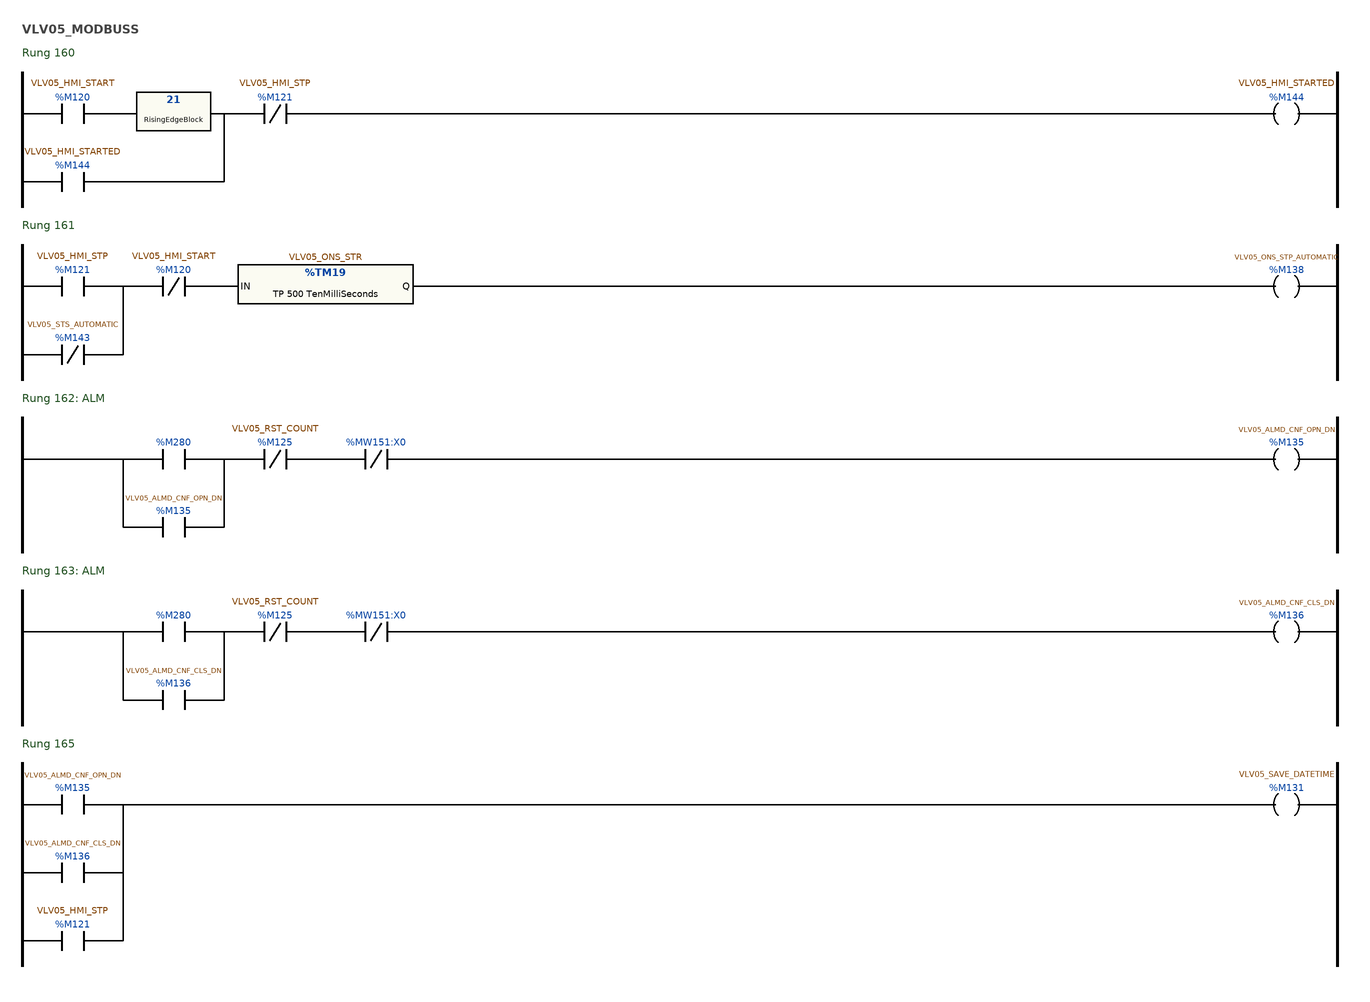
[picture p24: VLV05_MODBUSS, ladder]

// Rung 160
  LD %M120                (* VLV05_HMI_START *)
  RISING21
  OR %M144                (* VLV05_HMI_STARTED *)
  ANDN %M121              (* VLV05_HMI_STP *)
  ST %M144                (* VLV05_HMI_STARTED *)
  // as ST:
  //   VLV05_HMI_STARTED := (RISING(VLV05_HMI_START) OR VLV05_HMI_STARTED) AND NOT VLV05_HMI_STP;

// Rung 161
  BLK %TM19               (* VLV05_ONS_STR *)
  LD %M121                (* VLV05_HMI_STP *)
  ORN %M143               (* VLV05_STS_AUTOMATIC *)
  ANDN %M120              (* VLV05_HMI_START *)
  IN
  OUT_BLK
  LD Q
  ST %M138                (* VLV05_ONS_STP_AUTOMATIC *)
  END_BLK
  // as ST:
  //   VLV05_ONS_STR(IN := (VLV05_HMI_STP OR NOT VLV05_STS_AUTOMATIC) AND NOT VLV05_HMI_START);
  //   VLV05_ONS_STP_AUTOMATIC := VLV05_ONS_STR.Q;

// Rung 162: ALM
  LD 1
  AND( %M280
  OR %M135                (* VLV05_ALMD_CNF_OPN_DN *)
  )
  ANDN %M125              (* VLV05_RST_COUNT *)
  ANDN %MW151:X0
  ST %M135                (* VLV05_ALMD_CNF_OPN_DN *)
  // as ST:
  //   VLV05_ALMD_CNF_OPN_DN := (%M280 OR VLV05_ALMD_CNF_OPN_DN) AND NOT VLV05_RST_COUNT AND NOT %MW151:X0;

// Rung 163: ALM
  LD 1
  AND( %M280
  OR %M136                (* VLV05_ALMD_CNF_CLS_DN *)
  )
  ANDN %M125              (* VLV05_RST_COUNT *)
  ANDN %MW151:X0
  ST %M136                (* VLV05_ALMD_CNF_CLS_DN *)
  // as ST:
  //   VLV05_ALMD_CNF_CLS_DN := (%M280 OR VLV05_ALMD_CNF_CLS_DN) AND NOT VLV05_RST_COUNT AND NOT %MW151:X0;

// Rung 164
  LD 1
  MULTIFB
  LD 1
  AND %M21                (* HORARIOOFICINA_ACTIVE *)
  AND %M144               (* VLV05_HMI_STARTED *)
  ANDN %M135              (* VLV05_ALMD_CNF_OPN_DN *)
  ANDN %M136              (* VLV05_ALMD_CNF_CLS_DN *)
  AND %MW444:X0
  ANDN %M148              (* VLV05_TON_HR_DN *)
  ST %MW2509:X0
  LD %MW2509:X0
  ST %M143                (* VLV05_STS_AUTOMATIC *)
  BLK %TM47               (* VLV05_ONS_01 *)
  LD %MW2509:X0
  IN
  OUT_BLK
  LD Q
  ST %M126                (* VLV05_ONS_STS_AUTOMATIC *)
  END_BLK
  MULTIFB
  // as ST:
  //   %MW2509:X0 := HORARIOOFICINA_ACTIVE AND VLV05_HMI_STARTED AND NOT VLV05_ALMD_CNF_OPN_DN AND NOT VLV05_ALMD_CNF_CLS_DN AND %MW444:X0 AND NOT VLV05_TON_HR_DN;
  //   VLV05_STS_AUTOMATIC := %MW2509:X0;
  //   VLV05_ONS_01(IN := %MW2509:X0);
  //   VLV05_ONS_STS_AUTOMATIC := VLV05_ONS_01.Q;
  (* the ladder stored for this rung does not match its IL; not drawn *)

// Rung 165
  LD %M135                (* VLV05_ALMD_CNF_OPN_DN *)
  OR %M136                (* VLV05_ALMD_CNF_CLS_DN *)
  OR %M121                (* VLV05_HMI_STP *)
  ST %M131                (* VLV05_SAVE_DATETIME *)
  // as ST:
  //   VLV05_SAVE_DATETIME := VLV05_ALMD_CNF_OPN_DN OR VLV05_ALMD_CNF_CLS_DN OR VLV05_HMI_STP;

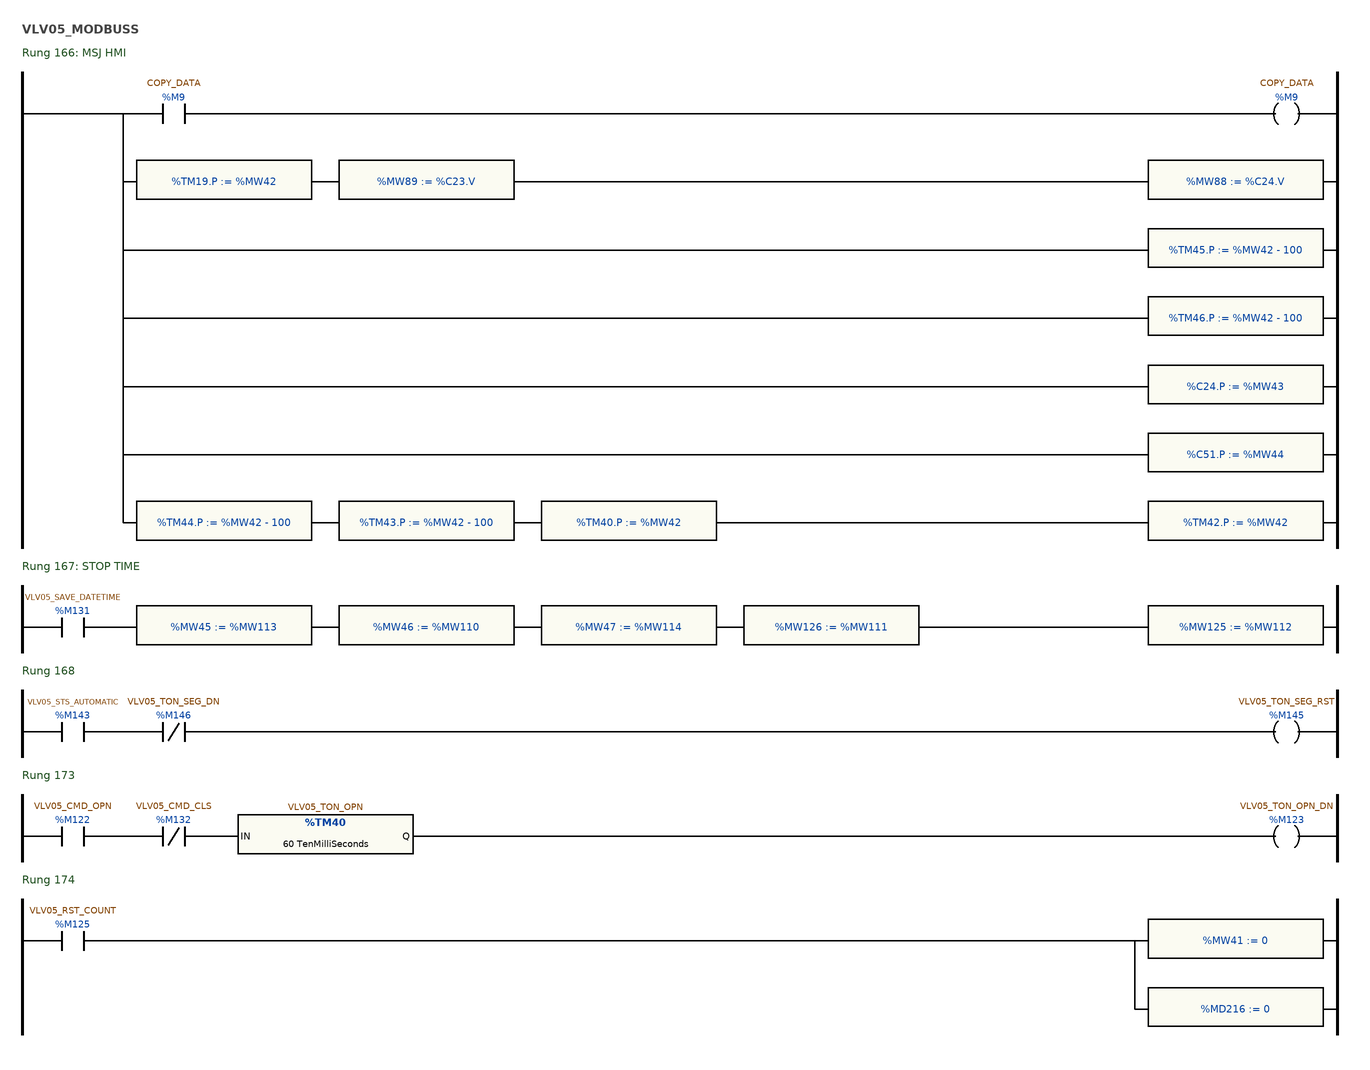

// Rung 166: MSJ HMI
  LD 1
  MPS
  AND %M9                 (* COPY_DATA *)
  ST %M9                  (* COPY_DATA *)
  MRD
  OPER [ %TM19.P := %MW42 ](* VLV05_ONS_STR, VLV05_T_CNF_PRESET *)
  OPER [ %MW89 := %C23.V ](* VLV05_CNT_MIN *)
  [ %MW88 := %C24.V ]     (* VLV05_CNT_HR *)
  MRD
  [ %TM45.P := %MW42 - 100 ](* VLV05_T_CNF_OPN, VLV05_T_CNF_PRESET *)
  MRD
  [ %TM46.P := %MW42 - 100 ](* VLV05_T_CNF_CLS, VLV05_T_CNF_PRESET *)
  MRD
  [ %C24.P := %MW43 ]     (* VLV05_CNT_HR, VLV05_CNF_HR_PRESET *)
  MRD
  [ %C51.P := %MW44 ]
  MPP
  OPER [ %TM44.P := %MW42 - 100 ](* VLV05_TON_ALMD_CNF_CLS, VLV05_T_CNF_PRESET *)
  OPER [ %TM43.P := %MW42 - 100 ](* VLV05_TON_ALMD_CNF_OPN, VLV05_T_CNF_PRESET *)
  OPER [ %TM40.P := %MW42 ](* VLV05_TON_OPN, VLV05_T_CNF_PRESET *)
  [ %TM42.P := %MW42 ]    (* VLV05_TON_CLS, VLV05_T_CNF_PRESET *)
  // as ST:
  //   COPY_DATA := COPY_DATA;
  //   VLV05_ONS_STR.P := VLV05_T_CNF_PRESET;
  //   %MW89 := VLV05_CNT_MIN.V;
  //   %MW88 := VLV05_CNT_HR.V;
  //   VLV05_T_CNF_OPN.P := VLV05_T_CNF_PRESET - 100;
  //   VLV05_T_CNF_CLS.P := VLV05_T_CNF_PRESET - 100;
  //   VLV05_CNT_HR.P := VLV05_CNF_HR_PRESET;
  //   %C51.P := %MW44;
  //   VLV05_TON_ALMD_CNF_CLS.P := VLV05_T_CNF_PRESET - 100;
  //   VLV05_TON_ALMD_CNF_OPN.P := VLV05_T_CNF_PRESET - 100;
  //   VLV05_TON_OPN.P := VLV05_T_CNF_PRESET;
  //   VLV05_TON_CLS.P := VLV05_T_CNF_PRESET;

// Rung 167: STOP TIME
  LD %M131                (* VLV05_SAVE_DATETIME *)
  OPER [ %MW45 := %MW113 ](* VLV05_RTC_HHMM, MONTH *)
  OPER [ %MW46 := %MW110 ](* VLV05_RTC_MMDD, DAY *)
  OPER [ %MW47 := %MW114 ](* VLV05_RTC_YY, YEAR *)
  OPER [ %MW126 := %MW111 ](* HOUR *)
  [ %MW125 := %MW112 ]    (* MINUTES *)
  // as ST:
  //   IF VLV05_SAVE_DATETIME THEN VLV05_RTC_HHMM := MONTH; END_IF;
  //   IF VLV05_SAVE_DATETIME THEN VLV05_RTC_MMDD := DAY; END_IF;
  //   IF VLV05_SAVE_DATETIME THEN VLV05_RTC_YY := YEAR; END_IF;
  //   IF VLV05_SAVE_DATETIME THEN %MW126 := HOUR; END_IF;
  //   IF VLV05_SAVE_DATETIME THEN %MW125 := MINUTES; END_IF;

// Rung 168
  LD %M143                (* VLV05_STS_AUTOMATIC *)
  ANDN %M146              (* VLV05_TON_SEG_DN *)
  ST %M145                (* VLV05_TON_SEG_RST *)
  // as ST:
  //   VLV05_TON_SEG_RST := VLV05_STS_AUTOMATIC AND NOT VLV05_TON_SEG_DN;

// Rung 169
  BLK %C24                (* VLV05_CNT_HR *)
  LD %M125                (* VLV05_RST_COUNT *)
  OR( %M21                (* HORARIOOFICINA_ACTIVE *)
  RISING22
  )
  R
  LD %M147                (* VLV05_TON_MIN_DN *)
  CU
  OUT_BLK
  LD D
  ST %M148                (* VLV05_TON_HR_DN *)
  END_BLK
  // as ST:
  //   VLV05_CNT_HR(RISING22 := HORARIOOFICINA_ACTIVE, R := VLV05_RST_COUNT OR HORARIOOFICINA_ACTIVE, CU := VLV05_TON_MIN_DN);
  //   VLV05_TON_HR_DN := VLV05_CNT_HR.D;
  (* the ladder stored for this rung does not match its IL; not drawn *)

// Rung 170
  BLK %C23                (* VLV05_CNT_MIN *)
  LD 1
  AND( %M125              (* VLV05_RST_COUNT *)
  OR %M147                (* VLV05_TON_MIN_DN *)
  )
  OR( %M21                (* HORARIOOFICINA_ACTIVE *)
  RISING23
  )
  R
  LD %M146                (* VLV05_TON_SEG_DN *)
  CU
  OUT_BLK
  LD D
  ST %M147                (* VLV05_TON_MIN_DN *)
  END_BLK
  // as ST:
  //   VLV05_CNT_MIN(RISING23 := HORARIOOFICINA_ACTIVE, R := VLV05_RST_COUNT OR VLV05_TON_MIN_DN OR HORARIOOFICINA_ACTIVE, CU := VLV05_TON_SEG_DN);
  //   VLV05_TON_MIN_DN := VLV05_CNT_MIN.D;
  (* the ladder stored for this rung does not match its IL; not drawn *)

// Rung 171
  LD 1
  MULTIFB
  LD 1
  ST %MW2509:X1
  BLK %TM41               (* VLV05_TON_SEG *)
  LD %MW2509:X1
  AND %M143               (* VLV05_STS_AUTOMATIC *)
  ANDN %M146              (* VLV05_TON_SEG_DN *)
  IN
  OUT_BLK
  LD Q
  ST %MW2509:X0
  END_BLK
  BLK %C22                (* VLV05_CNT_SEG *)
  LD %MW2509:X1
  AND( %M125              (* VLV05_RST_COUNT *)
  OR %M146                (* VLV05_TON_SEG_DN *)
  )
  R
  LD %MW2509:X0
  CU
  OUT_BLK
  LD D
  ST %M146                (* VLV05_TON_SEG_DN *)
  END_BLK
  MULTIFB
  // as ST:
  //   %MW2509:X1 := TRUE;
  //   VLV05_TON_SEG(IN := %MW2509:X1 AND VLV05_STS_AUTOMATIC AND NOT VLV05_TON_SEG_DN);
  //   %MW2509:X0 := VLV05_TON_SEG.Q;
  //   VLV05_CNT_SEG(R := %MW2509:X1 AND (VLV05_RST_COUNT OR VLV05_TON_SEG_DN), CU := %MW2509:X0);
  //   VLV05_TON_SEG_DN := VLV05_CNT_SEG.D;
  (* the ladder stored for this rung does not match its IL; not drawn *)

// Rung 172
  LD 1
  MULTIFB
  LD 1
  AND %M143               (* VLV05_STS_AUTOMATIC *)
  AND( %M126              (* VLV05_ONS_STS_AUTOMATIC *)
  OR %M133                (* VLV05_TON_CLS_DN *)
  OR %M122                (* VLV05_CMD_OPN *)
  )
  ANDN %M121              (* VLV05_HMI_STP *)
  ANDN %M123              (* VLV05_TON_OPN_DN *)
  OPER [ %MW90 := %MW9 ]
  ST %MW2509:X0
  LD %MW2509:X0
  ST %M122                (* VLV05_CMD_OPN *)
  BLK %TM90
  LD %MW2509:X0
  IN
  OUT_BLK
  LD Q
  ST %M310
  END_BLK
  MULTIFB
  // as ST:
  //   IF VLV05_STS_AUTOMATIC AND (VLV05_ONS_STS_AUTOMATIC OR VLV05_TON_CLS_DN OR VLV05_CMD_OPN) AND NOT VLV05_HMI_STP AND NOT VLV05_TON_OPN_DN THEN %MW90 := %MW9; END_IF;
  //   %MW2509:X0 := VLV05_STS_AUTOMATIC AND (VLV05_ONS_STS_AUTOMATIC OR VLV05_TON_CLS_DN OR VLV05_CMD_OPN) AND NOT VLV05_HMI_STP AND NOT VLV05_TON_OPN_DN;
  //   VLV05_CMD_OPN := %MW2509:X0;
  //   %TM90(IN := %MW2509:X0);
  //   %M310 := %TM90.Q;
  (* the ladder stored for this rung does not match its IL; not drawn *)

// Rung 173
  BLK %TM40               (* VLV05_TON_OPN *)
  LD %M122                (* VLV05_CMD_OPN *)
  ANDN %M132              (* VLV05_CMD_CLS *)
  IN
  OUT_BLK
  LD Q
  ST %M123                (* VLV05_TON_OPN_DN *)
  END_BLK
  // as ST:
  //   VLV05_TON_OPN(IN := VLV05_CMD_OPN AND NOT VLV05_CMD_CLS);
  //   VLV05_TON_OPN_DN := VLV05_TON_OPN.Q;

// Rung 174
  LD %M125                (* VLV05_RST_COUNT *)
  [ %MW41 := 0 ]          (* VLV05_CNT_OPN_ACC *)
  [ %MD216 := 0 ]         (* VLV05_CNT_OPN_ACC2 *)
  // as ST:
  //   IF VLV05_RST_COUNT THEN VLV05_CNT_OPN_ACC := 0; END_IF;
  //   IF VLV05_RST_COUNT THEN VLV05_CNT_OPN_ACC2 := 0; END_IF;

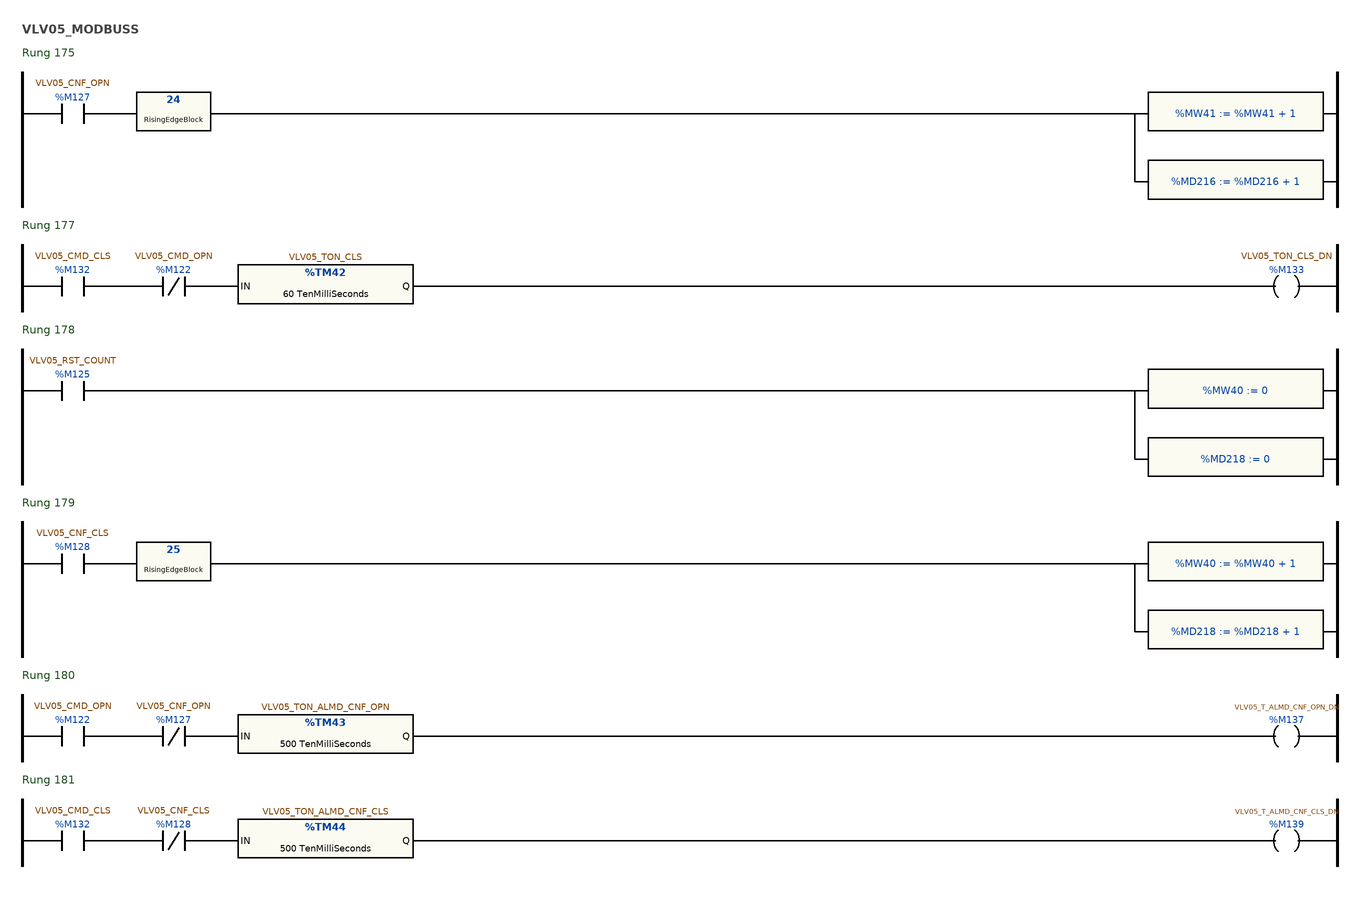

// Rung 175
  LD %M127                (* VLV05_CNF_OPN *)
  RISING24
  [ %MW41 := %MW41 + 1 ]  (* VLV05_CNT_OPN_ACC, VLV05_CNT_OPN_ACC *)
  [ %MD216 := %MD216 + 1 ](* VLV05_CNT_OPN_ACC2, VLV05_CNT_OPN_ACC2 *)
  // as ST:
  //   IF RISING(VLV05_CNF_OPN) THEN VLV05_CNT_OPN_ACC := VLV05_CNT_OPN_ACC + 1; END_IF;
  //   IF RISING(VLV05_CNF_OPN) THEN VLV05_CNT_OPN_ACC2 := VLV05_CNT_OPN_ACC2 + 1; END_IF;

// Rung 176
  LD 1
  MULTIFB
  LD 1
  AND %M143               (* VLV05_STS_AUTOMATIC *)
  AND( %M123              (* VLV05_TON_OPN_DN *)
  OR %M132                (* VLV05_CMD_CLS *)
  )
  ANDN %M121              (* VLV05_HMI_STP *)
  ANDN %M133              (* VLV05_TON_CLS_DN *)
  OR %M138                (* VLV05_ONS_STP_AUTOMATIC *)
  OPER [ %MW90 := %MW44 ]
  ST %MW2509:X0
  LD %MW2509:X0
  ST %M132                (* VLV05_CMD_CLS *)
  BLK %TM96
  LD %MW2509:X0
  IN
  OUT_BLK
  LD Q
  ST %M311
  END_BLK
  MULTIFB
  // as ST:
  //   IF VLV05_STS_AUTOMATIC AND (VLV05_TON_OPN_DN OR VLV05_CMD_CLS) AND NOT VLV05_HMI_STP AND NOT VLV05_TON_CLS_DN OR VLV05_ONS_STP_AUTOMATIC THEN %MW90 := %MW44; END_IF;
  //   %MW2509:X0 := VLV05_STS_AUTOMATIC AND (VLV05_TON_OPN_DN OR VLV05_CMD_CLS) AND NOT VLV05_HMI_STP AND NOT VLV05_TON_CLS_DN OR VLV05_ONS_STP_AUTOMATIC;
  //   VLV05_CMD_CLS := %MW2509:X0;
  //   %TM96(IN := %MW2509:X0);
  //   %M311 := %TM96.Q;
  (* the ladder stored for this rung does not match its IL; not drawn *)

// Rung 177
  BLK %TM42               (* VLV05_TON_CLS *)
  LD %M132                (* VLV05_CMD_CLS *)
  ANDN %M122              (* VLV05_CMD_OPN *)
  IN
  OUT_BLK
  LD Q
  ST %M133                (* VLV05_TON_CLS_DN *)
  END_BLK
  // as ST:
  //   VLV05_TON_CLS(IN := VLV05_CMD_CLS AND NOT VLV05_CMD_OPN);
  //   VLV05_TON_CLS_DN := VLV05_TON_CLS.Q;

// Rung 178
  LD %M125                (* VLV05_RST_COUNT *)
  [ %MW40 := 0 ]          (* VLV05_CNT_CLS_ACC *)
  [ %MD218 := 0 ]         (* VLV05_CNT_CLS_ACC2 *)
  // as ST:
  //   IF VLV05_RST_COUNT THEN VLV05_CNT_CLS_ACC := 0; END_IF;
  //   IF VLV05_RST_COUNT THEN VLV05_CNT_CLS_ACC2 := 0; END_IF;

// Rung 179
  LD %M128                (* VLV05_CNF_CLS *)
  RISING25
  [ %MW40 := %MW40 + 1 ]  (* VLV05_CNT_CLS_ACC, VLV05_CNT_CLS_ACC *)
  [ %MD218 := %MD218 + 1 ](* VLV05_CNT_CLS_ACC2, VLV05_CNT_CLS_ACC2 *)
  // as ST:
  //   IF RISING(VLV05_CNF_CLS) THEN VLV05_CNT_CLS_ACC := VLV05_CNT_CLS_ACC + 1; END_IF;
  //   IF RISING(VLV05_CNF_CLS) THEN VLV05_CNT_CLS_ACC2 := VLV05_CNT_CLS_ACC2 + 1; END_IF;

// Rung 180
  BLK %TM43               (* VLV05_TON_ALMD_CNF_OPN *)
  LD %M122                (* VLV05_CMD_OPN *)
  ANDN %M127              (* VLV05_CNF_OPN *)
  IN
  OUT_BLK
  LD Q
  ST %M137                (* VLV05_T_ALMD_CNF_OPN_DN *)
  END_BLK
  // as ST:
  //   VLV05_TON_ALMD_CNF_OPN(IN := VLV05_CMD_OPN AND NOT VLV05_CNF_OPN);
  //   VLV05_T_ALMD_CNF_OPN_DN := VLV05_TON_ALMD_CNF_OPN.Q;

// Rung 181
  BLK %TM44               (* VLV05_TON_ALMD_CNF_CLS *)
  LD %M132                (* VLV05_CMD_CLS *)
  ANDN %M128              (* VLV05_CNF_CLS *)
  IN
  OUT_BLK
  LD Q
  ST %M139                (* VLV05_T_ALMD_CNF_CLS_DN *)
  END_BLK
  // as ST:
  //   VLV05_TON_ALMD_CNF_CLS(IN := VLV05_CMD_CLS AND NOT VLV05_CNF_CLS);
  //   VLV05_T_ALMD_CNF_CLS_DN := VLV05_TON_ALMD_CNF_CLS.Q;

POU VLV06_MODBUSS
  (* SectionNumber=7 *)

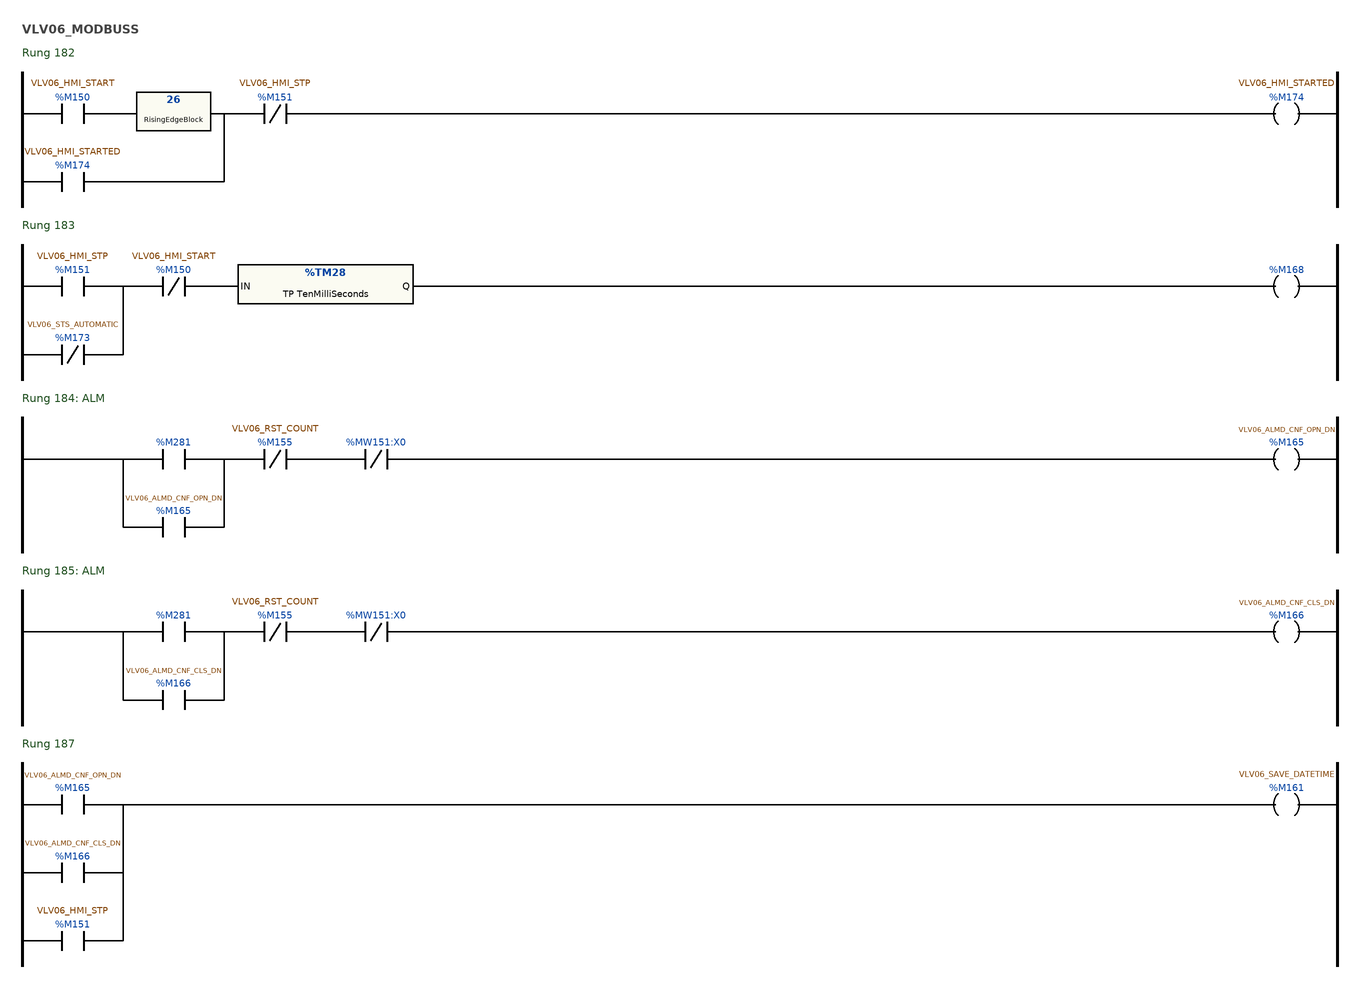

// Rung 182
  LD %M150                (* VLV06_HMI_START *)
  RISING26
  OR %M174                (* VLV06_HMI_STARTED *)
  ANDN %M151              (* VLV06_HMI_STP *)
  ST %M174                (* VLV06_HMI_STARTED *)
  // as ST:
  //   VLV06_HMI_STARTED := (RISING(VLV06_HMI_START) OR VLV06_HMI_STARTED) AND NOT VLV06_HMI_STP;

// Rung 183
  BLK %TM28
  LD %M151                (* VLV06_HMI_STP *)
  ORN %M173               (* VLV06_STS_AUTOMATIC *)
  ANDN %M150              (* VLV06_HMI_START *)
  IN
  OUT_BLK
  LD Q
  ST %M168
  END_BLK
  // as ST:
  //   %TM28(IN := (VLV06_HMI_STP OR NOT VLV06_STS_AUTOMATIC) AND NOT VLV06_HMI_START);
  //   %M168 := %TM28.Q;

// Rung 184: ALM
  LD 1
  AND( %M281
  OR %M165                (* VLV06_ALMD_CNF_OPN_DN *)
  )
  ANDN %M155              (* VLV06_RST_COUNT *)
  ANDN %MW151:X0
  ST %M165                (* VLV06_ALMD_CNF_OPN_DN *)
  // as ST:
  //   VLV06_ALMD_CNF_OPN_DN := (%M281 OR VLV06_ALMD_CNF_OPN_DN) AND NOT VLV06_RST_COUNT AND NOT %MW151:X0;

// Rung 185: ALM
  LD 1
  AND( %M281
  OR %M166                (* VLV06_ALMD_CNF_CLS_DN *)
  )
  ANDN %M155              (* VLV06_RST_COUNT *)
  ANDN %MW151:X0
  ST %M166                (* VLV06_ALMD_CNF_CLS_DN *)
  // as ST:
  //   VLV06_ALMD_CNF_CLS_DN := (%M281 OR VLV06_ALMD_CNF_CLS_DN) AND NOT VLV06_RST_COUNT AND NOT %MW151:X0;

// Rung 186
  LD 1
  MULTIFB
  LD 1
  AND %M21                (* HORARIOOFICINA_ACTIVE *)
  AND %M174               (* VLV06_HMI_STARTED *)
  ANDN %M165              (* VLV06_ALMD_CNF_OPN_DN *)
  ANDN %M166              (* VLV06_ALMD_CNF_CLS_DN *)
  AND %MW444:X0
  ANDN %M168
  ANDN %M178              (* VLV06_TON_HR_DN *)
  ST %MW2509:X0
  LD %MW2509:X0
  ST %M173                (* VLV06_STS_AUTOMATIC *)
  BLK %TM57               (* VLV06_ONS *)
  LD %MW2509:X0
  IN
  OUT_BLK
  LD Q
  ST %M156                (* VLV06_ONS_STS_AUTOMATIC *)
  END_BLK
  MULTIFB
  // as ST:
  //   %MW2509:X0 := HORARIOOFICINA_ACTIVE AND VLV06_HMI_STARTED AND NOT VLV06_ALMD_CNF_OPN_DN AND NOT VLV06_ALMD_CNF_CLS_DN AND %MW444:X0 AND NOT %M168 AND NOT VLV06_TON_HR_DN;
  //   VLV06_STS_AUTOMATIC := %MW2509:X0;
  //   VLV06_ONS(IN := %MW2509:X0);
  //   VLV06_ONS_STS_AUTOMATIC := VLV06_ONS.Q;
  (* the ladder stored for this rung does not match its IL; not drawn *)

// Rung 187
  LD %M165                (* VLV06_ALMD_CNF_OPN_DN *)
  OR %M166                (* VLV06_ALMD_CNF_CLS_DN *)
  OR %M151                (* VLV06_HMI_STP *)
  ST %M161                (* VLV06_SAVE_DATETIME *)
  // as ST:
  //   VLV06_SAVE_DATETIME := VLV06_ALMD_CNF_OPN_DN OR VLV06_ALMD_CNF_CLS_DN OR VLV06_HMI_STP;

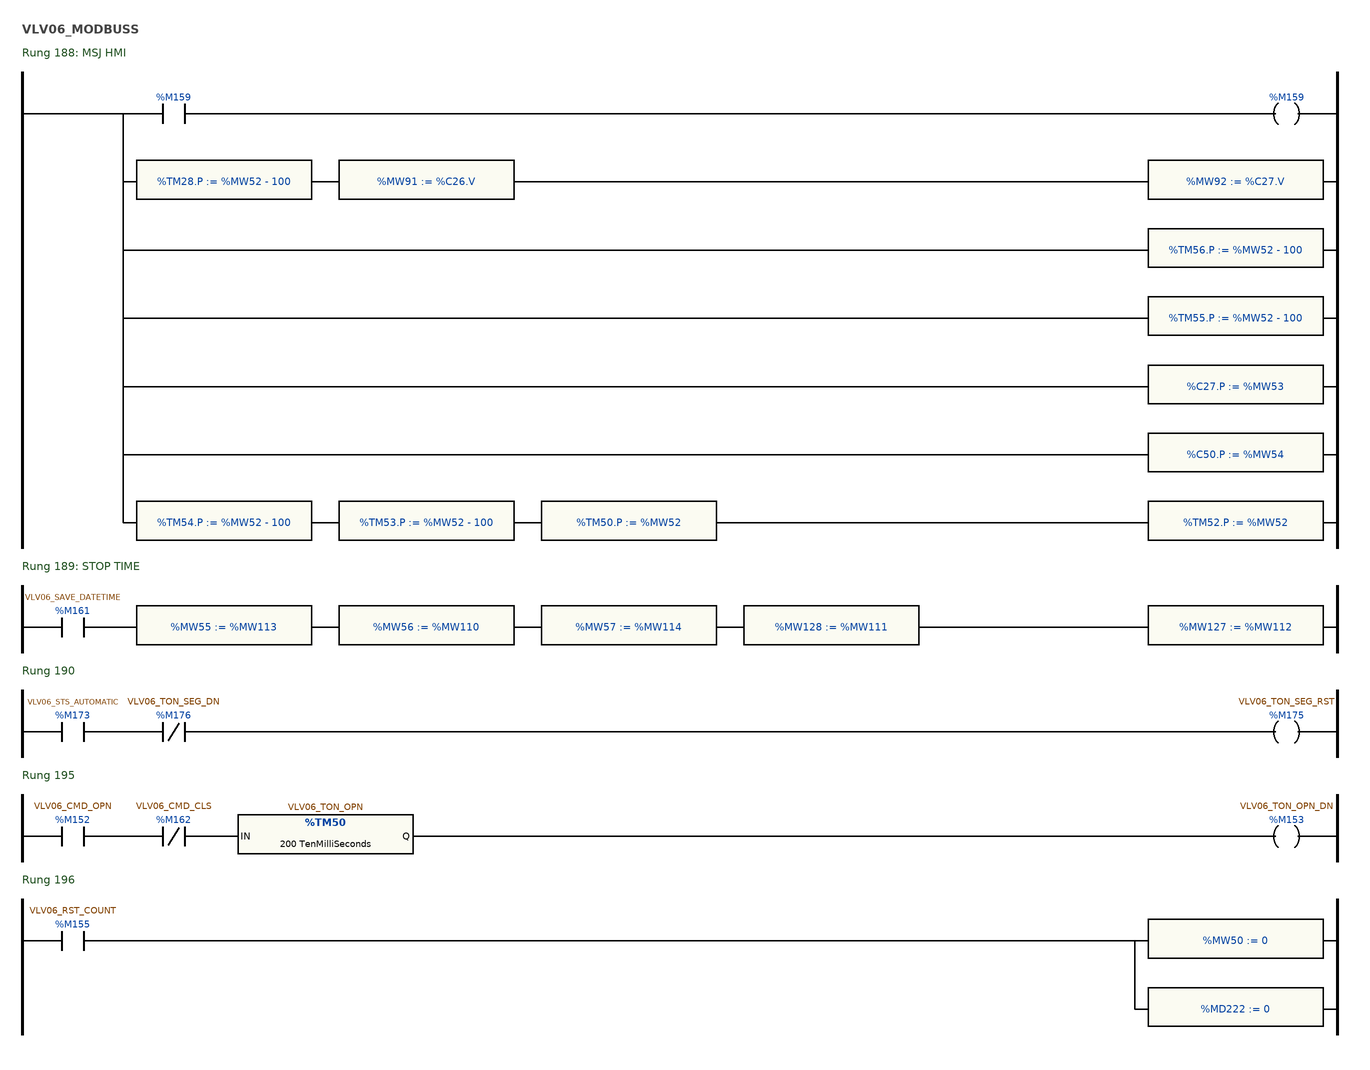

// Rung 188: MSJ HMI
  LD 1
  MPS
  AND %M159
  ST %M159
  MRD
  OPER [ %TM28.P := %MW52 - 100 ](* VLV06_T_CNF_PRESET *)
  OPER [ %MW91 := %C26.V ](* VLV06_CNT_MIN *)
  [ %MW92 := %C27.V ]     (* VLV06_CNT_HR *)
  MRD
  [ %TM56.P := %MW52 - 100 ](* VLV06_T_CNF_CLS, VLV06_T_CNF_PRESET *)
  MRD
  [ %TM55.P := %MW52 - 100 ](* VLV06_T_CNF_OPN, VLV06_T_CNF_PRESET *)
  MRD
  [ %C27.P := %MW53 ]     (* VLV06_CNT_HR, VLV06_CNF_HR_PRESET *)
  MRD
  [ %C50.P := %MW54 ]
  MPP
  OPER [ %TM54.P := %MW52 - 100 ](* VLV06_TON_ALMD_CNF_CLS, VLV06_T_CNF_PRESET *)
  OPER [ %TM53.P := %MW52 - 100 ](* VLV06_TON_ALMD_CNF_OPN, VLV06_T_CNF_PRESET *)
  OPER [ %TM50.P := %MW52 ](* VLV06_TON_OPN, VLV06_T_CNF_PRESET *)
  [ %TM52.P := %MW52 ]    (* VLV06_TON_CLS, VLV06_T_CNF_PRESET *)
  // as ST:
  //   %M159 := %M159;
  //   %TM28.P := VLV06_T_CNF_PRESET - 100;
  //   %MW91 := VLV06_CNT_MIN.V;
  //   %MW92 := VLV06_CNT_HR.V;
  //   VLV06_T_CNF_CLS.P := VLV06_T_CNF_PRESET - 100;
  //   VLV06_T_CNF_OPN.P := VLV06_T_CNF_PRESET - 100;
  //   VLV06_CNT_HR.P := VLV06_CNF_HR_PRESET;
  //   %C50.P := %MW54;
  //   VLV06_TON_ALMD_CNF_CLS.P := VLV06_T_CNF_PRESET - 100;
  //   VLV06_TON_ALMD_CNF_OPN.P := VLV06_T_CNF_PRESET - 100;
  //   VLV06_TON_OPN.P := VLV06_T_CNF_PRESET;
  //   VLV06_TON_CLS.P := VLV06_T_CNF_PRESET;

// Rung 189: STOP TIME
  LD %M161                (* VLV06_SAVE_DATETIME *)
  OPER [ %MW55 := %MW113 ](* VLV06_RTC_HHMM, MONTH *)
  OPER [ %MW56 := %MW110 ](* VLV06_RTC_MMDD, DAY *)
  OPER [ %MW57 := %MW114 ](* VLV06_RTC_YY, YEAR *)
  OPER [ %MW128 := %MW111 ](* HOUR *)
  [ %MW127 := %MW112 ]    (* MINUTES *)
  // as ST:
  //   IF VLV06_SAVE_DATETIME THEN VLV06_RTC_HHMM := MONTH; END_IF;
  //   IF VLV06_SAVE_DATETIME THEN VLV06_RTC_MMDD := DAY; END_IF;
  //   IF VLV06_SAVE_DATETIME THEN VLV06_RTC_YY := YEAR; END_IF;
  //   IF VLV06_SAVE_DATETIME THEN %MW128 := HOUR; END_IF;
  //   IF VLV06_SAVE_DATETIME THEN %MW127 := MINUTES; END_IF;

// Rung 190
  LD %M173                (* VLV06_STS_AUTOMATIC *)
  ANDN %M176              (* VLV06_TON_SEG_DN *)
  ST %M175                (* VLV06_TON_SEG_RST *)
  // as ST:
  //   VLV06_TON_SEG_RST := VLV06_STS_AUTOMATIC AND NOT VLV06_TON_SEG_DN;

// Rung 191
  BLK %C27                (* VLV06_CNT_HR *)
  LD %M155                (* VLV06_RST_COUNT *)
  OR( %M21                (* HORARIOOFICINA_ACTIVE *)
  RISING27
  )
  R
  LD %M177                (* VLV06_TON_MIN_DN *)
  CU
  OUT_BLK
  LD D
  ST %M178                (* VLV06_TON_HR_DN *)
  END_BLK
  // as ST:
  //   VLV06_CNT_HR(RISING27 := HORARIOOFICINA_ACTIVE, R := VLV06_RST_COUNT OR HORARIOOFICINA_ACTIVE, CU := VLV06_TON_MIN_DN);
  //   VLV06_TON_HR_DN := VLV06_CNT_HR.D;
  (* the ladder stored for this rung does not match its IL; not drawn *)

// Rung 192
  BLK %C26                (* VLV06_CNT_MIN *)
  LD 1
  AND( %M155              (* VLV06_RST_COUNT *)
  OR %M177                (* VLV06_TON_MIN_DN *)
  )
  OR( %M21                (* HORARIOOFICINA_ACTIVE *)
  RISING28
  )
  R
  LD %M176                (* VLV06_TON_SEG_DN *)
  CU
  OUT_BLK
  LD D
  ST %M177                (* VLV06_TON_MIN_DN *)
  END_BLK
  // as ST:
  //   VLV06_CNT_MIN(RISING28 := HORARIOOFICINA_ACTIVE, R := VLV06_RST_COUNT OR VLV06_TON_MIN_DN OR HORARIOOFICINA_ACTIVE, CU := VLV06_TON_SEG_DN);
  //   VLV06_TON_MIN_DN := VLV06_CNT_MIN.D;
  (* the ladder stored for this rung does not match its IL; not drawn *)

// Rung 193
  LD 1
  MULTIFB
  LD 1
  ST %MW2509:X1
  BLK %TM51               (* VLV06_TON_SEG *)
  LD %MW2509:X1
  AND %M173               (* VLV06_STS_AUTOMATIC *)
  ANDN %M176              (* VLV06_TON_SEG_DN *)
  IN
  OUT_BLK
  LD Q
  ST %MW2509:X0
  END_BLK
  BLK %C25                (* VLV06_CNT_SEG *)
  LD %MW2509:X1
  AND( %M155              (* VLV06_RST_COUNT *)
  OR %M176                (* VLV06_TON_SEG_DN *)
  )
  R
  LD %MW2509:X0
  CU
  OUT_BLK
  LD D
  ST %M176                (* VLV06_TON_SEG_DN *)
  END_BLK
  MULTIFB
  // as ST:
  //   %MW2509:X1 := TRUE;
  //   VLV06_TON_SEG(IN := %MW2509:X1 AND VLV06_STS_AUTOMATIC AND NOT VLV06_TON_SEG_DN);
  //   %MW2509:X0 := VLV06_TON_SEG.Q;
  //   VLV06_CNT_SEG(R := %MW2509:X1 AND (VLV06_RST_COUNT OR VLV06_TON_SEG_DN), CU := %MW2509:X0);
  //   VLV06_TON_SEG_DN := VLV06_CNT_SEG.D;
  (* the ladder stored for this rung does not match its IL; not drawn *)

// Rung 194
  LD 1
  MULTIFB
  LD 1
  AND %M173               (* VLV06_STS_AUTOMATIC *)
  AND( %M156              (* VLV06_ONS_STS_AUTOMATIC *)
  OR %M163                (* VLV06_TON_CLS_DN *)
  OR %M152                (* VLV06_CMD_OPN *)
  )
  ANDN %M151              (* VLV06_HMI_STP *)
  ANDN %M153              (* VLV06_TON_OPN_DN *)
  OPER [ %MW100 := %MW58 ]
  ST %MW2509:X0
  LD %MW2509:X0
  ST %M152                (* VLV06_CMD_OPN *)
  BLK %TM87
  LD %MW2509:X0
  IN
  OUT_BLK
  LD Q
  ST %M313
  END_BLK
  MULTIFB
  // as ST:
  //   IF VLV06_STS_AUTOMATIC AND (VLV06_ONS_STS_AUTOMATIC OR VLV06_TON_CLS_DN OR VLV06_CMD_OPN) AND NOT VLV06_HMI_STP AND NOT VLV06_TON_OPN_DN THEN %MW100 := %MW58; END_IF;
  //   %MW2509:X0 := VLV06_STS_AUTOMATIC AND (VLV06_ONS_STS_AUTOMATIC OR VLV06_TON_CLS_DN OR VLV06_CMD_OPN) AND NOT VLV06_HMI_STP AND NOT VLV06_TON_OPN_DN;
  //   VLV06_CMD_OPN := %MW2509:X0;
  //   %TM87(IN := %MW2509:X0);
  //   %M313 := %TM87.Q;
  (* the ladder stored for this rung does not match its IL; not drawn *)

// Rung 195
  BLK %TM50               (* VLV06_TON_OPN *)
  LD %M152                (* VLV06_CMD_OPN *)
  ANDN %M162              (* VLV06_CMD_CLS *)
  IN
  OUT_BLK
  LD Q
  ST %M153                (* VLV06_TON_OPN_DN *)
  END_BLK
  // as ST:
  //   VLV06_TON_OPN(IN := VLV06_CMD_OPN AND NOT VLV06_CMD_CLS);
  //   VLV06_TON_OPN_DN := VLV06_TON_OPN.Q;

// Rung 196
  LD %M155                (* VLV06_RST_COUNT *)
  [ %MW50 := 0 ]          (* VLV06_CNT_CLS_ACC *)
  [ %MD222 := 0 ]         (* VLV06_CNT_CLS_ACC2 *)
  // as ST:
  //   IF VLV06_RST_COUNT THEN VLV06_CNT_CLS_ACC := 0; END_IF;
  //   IF VLV06_RST_COUNT THEN VLV06_CNT_CLS_ACC2 := 0; END_IF;

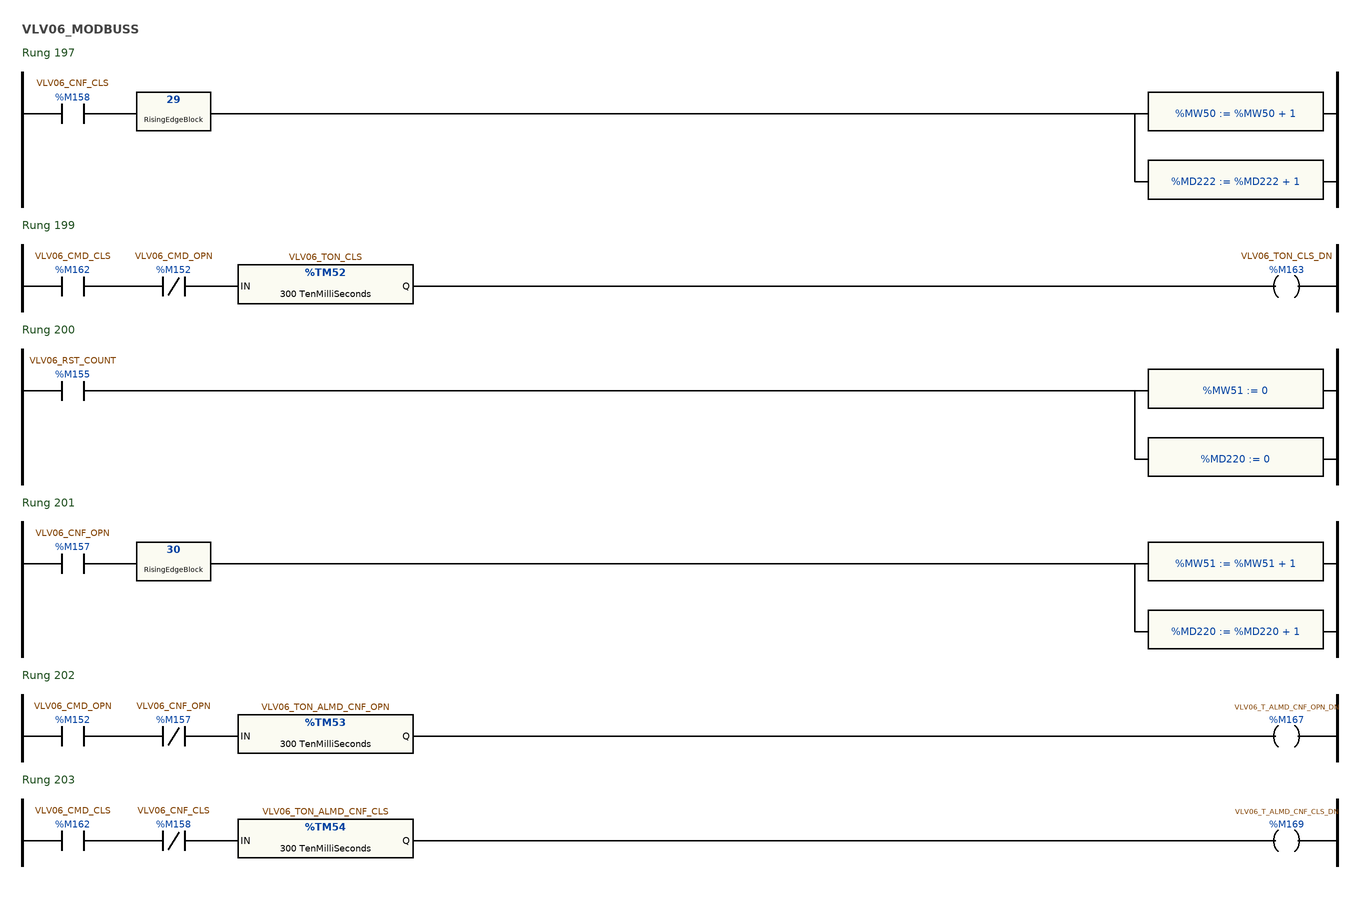

// Rung 197
  LD %M158                (* VLV06_CNF_CLS *)
  RISING29
  [ %MW50 := %MW50 + 1 ]  (* VLV06_CNT_CLS_ACC, VLV06_CNT_CLS_ACC *)
  [ %MD222 := %MD222 + 1 ](* VLV06_CNT_CLS_ACC2, VLV06_CNT_CLS_ACC2 *)
  // as ST:
  //   IF RISING(VLV06_CNF_CLS) THEN VLV06_CNT_CLS_ACC := VLV06_CNT_CLS_ACC + 1; END_IF;
  //   IF RISING(VLV06_CNF_CLS) THEN VLV06_CNT_CLS_ACC2 := VLV06_CNT_CLS_ACC2 + 1; END_IF;

// Rung 198
  LD 1
  MULTIFB
  LD 1
  AND %M173               (* VLV06_STS_AUTOMATIC *)
  AND( %M153              (* VLV06_TON_OPN_DN *)
  OR %M162                (* VLV06_CMD_CLS *)
  )
  ANDN %M151              (* VLV06_HMI_STP *)
  ANDN %M163              (* VLV06_TON_CLS_DN *)
  OR %M168
  OPER [ %MW100 := %MW54 ]
  ST %MW2509:X0
  LD %MW2509:X0
  ST %M162                (* VLV06_CMD_CLS *)
  BLK %TM91
  LD %MW2509:X0
  IN
  OUT_BLK
  LD Q
  ST %M312
  END_BLK
  MULTIFB
  // as ST:
  //   IF VLV06_STS_AUTOMATIC AND (VLV06_TON_OPN_DN OR VLV06_CMD_CLS) AND NOT VLV06_HMI_STP AND NOT VLV06_TON_CLS_DN OR %M168 THEN %MW100 := %MW54; END_IF;
  //   %MW2509:X0 := VLV06_STS_AUTOMATIC AND (VLV06_TON_OPN_DN OR VLV06_CMD_CLS) AND NOT VLV06_HMI_STP AND NOT VLV06_TON_CLS_DN OR %M168;
  //   VLV06_CMD_CLS := %MW2509:X0;
  //   %TM91(IN := %MW2509:X0);
  //   %M312 := %TM91.Q;
  (* the ladder stored for this rung does not match its IL; not drawn *)

// Rung 199
  BLK %TM52               (* VLV06_TON_CLS *)
  LD %M162                (* VLV06_CMD_CLS *)
  ANDN %M152              (* VLV06_CMD_OPN *)
  IN
  OUT_BLK
  LD Q
  ST %M163                (* VLV06_TON_CLS_DN *)
  END_BLK
  // as ST:
  //   VLV06_TON_CLS(IN := VLV06_CMD_CLS AND NOT VLV06_CMD_OPN);
  //   VLV06_TON_CLS_DN := VLV06_TON_CLS.Q;

// Rung 200
  LD %M155                (* VLV06_RST_COUNT *)
  [ %MW51 := 0 ]          (* VLV06_CNT_OPN_ACC *)
  [ %MD220 := 0 ]         (* VLV06_CNT_OPN_ACC2 *)
  // as ST:
  //   IF VLV06_RST_COUNT THEN VLV06_CNT_OPN_ACC := 0; END_IF;
  //   IF VLV06_RST_COUNT THEN VLV06_CNT_OPN_ACC2 := 0; END_IF;

// Rung 201
  LD %M157                (* VLV06_CNF_OPN *)
  RISING30
  [ %MW51 := %MW51 + 1 ]  (* VLV06_CNT_OPN_ACC, VLV06_CNT_OPN_ACC *)
  [ %MD220 := %MD220 + 1 ](* VLV06_CNT_OPN_ACC2, VLV06_CNT_OPN_ACC2 *)
  // as ST:
  //   IF RISING(VLV06_CNF_OPN) THEN VLV06_CNT_OPN_ACC := VLV06_CNT_OPN_ACC + 1; END_IF;
  //   IF RISING(VLV06_CNF_OPN) THEN VLV06_CNT_OPN_ACC2 := VLV06_CNT_OPN_ACC2 + 1; END_IF;

// Rung 202
  BLK %TM53               (* VLV06_TON_ALMD_CNF_OPN *)
  LD %M152                (* VLV06_CMD_OPN *)
  ANDN %M157              (* VLV06_CNF_OPN *)
  IN
  OUT_BLK
  LD Q
  ST %M167                (* VLV06_T_ALMD_CNF_OPN_DN *)
  END_BLK
  // as ST:
  //   VLV06_TON_ALMD_CNF_OPN(IN := VLV06_CMD_OPN AND NOT VLV06_CNF_OPN);
  //   VLV06_T_ALMD_CNF_OPN_DN := VLV06_TON_ALMD_CNF_OPN.Q;

// Rung 203
  BLK %TM54               (* VLV06_TON_ALMD_CNF_CLS *)
  LD %M162                (* VLV06_CMD_CLS *)
  ANDN %M158              (* VLV06_CNF_CLS *)
  IN
  OUT_BLK
  LD Q
  ST %M169                (* VLV06_T_ALMD_CNF_CLS_DN *)
  END_BLK
  // as ST:
  //   VLV06_TON_ALMD_CNF_CLS(IN := VLV06_CMD_CLS AND NOT VLV06_CNF_CLS);
  //   VLV06_T_ALMD_CNF_CLS_DN := VLV06_TON_ALMD_CNF_CLS.Q;

POU VLV07_CALENDAR
  (* SectionNumber=8 *)

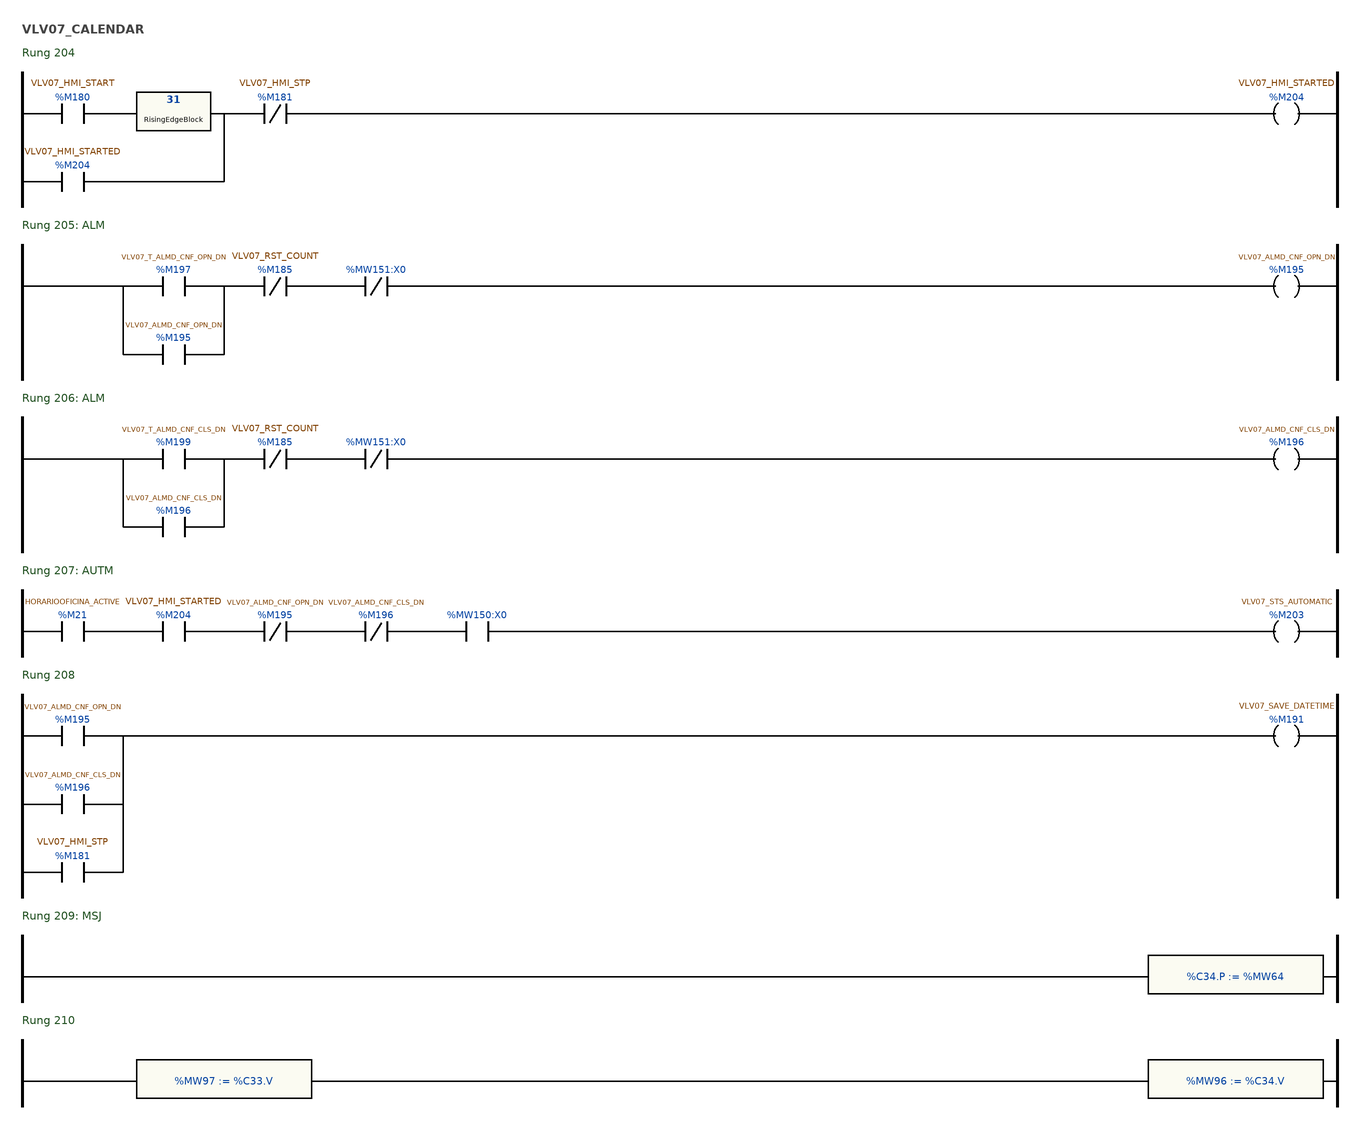

// Rung 204
  LD %M180                (* VLV07_HMI_START *)
  RISING31
  OR %M204                (* VLV07_HMI_STARTED *)
  ANDN %M181              (* VLV07_HMI_STP *)
  ST %M204                (* VLV07_HMI_STARTED *)
  // as ST:
  //   VLV07_HMI_STARTED := (RISING(VLV07_HMI_START) OR VLV07_HMI_STARTED) AND NOT VLV07_HMI_STP;

// Rung 205: ALM
  LD 1
  AND( %M197              (* VLV07_T_ALMD_CNF_OPN_DN *)
  OR %M195                (* VLV07_ALMD_CNF_OPN_DN *)
  )
  ANDN %M185              (* VLV07_RST_COUNT *)
  ANDN %MW151:X0
  ST %M195                (* VLV07_ALMD_CNF_OPN_DN *)
  // as ST:
  //   VLV07_ALMD_CNF_OPN_DN := (VLV07_T_ALMD_CNF_OPN_DN OR VLV07_ALMD_CNF_OPN_DN) AND NOT VLV07_RST_COUNT AND NOT %MW151:X0;

// Rung 206: ALM
  LD 1
  AND( %M199              (* VLV07_T_ALMD_CNF_CLS_DN *)
  OR %M196                (* VLV07_ALMD_CNF_CLS_DN *)
  )
  ANDN %M185              (* VLV07_RST_COUNT *)
  ANDN %MW151:X0
  ST %M196                (* VLV07_ALMD_CNF_CLS_DN *)
  // as ST:
  //   VLV07_ALMD_CNF_CLS_DN := (VLV07_T_ALMD_CNF_CLS_DN OR VLV07_ALMD_CNF_CLS_DN) AND NOT VLV07_RST_COUNT AND NOT %MW151:X0;

// Rung 207: AUTM
  LD %M21                 (* HORARIOOFICINA_ACTIVE *)
  AND %M204               (* VLV07_HMI_STARTED *)
  ANDN %M195              (* VLV07_ALMD_CNF_OPN_DN *)
  ANDN %M196              (* VLV07_ALMD_CNF_CLS_DN *)
  AND %MW150:X0
  ST %M203                (* VLV07_STS_AUTOMATIC *)
  // as ST:
  //   VLV07_STS_AUTOMATIC := HORARIOOFICINA_ACTIVE AND VLV07_HMI_STARTED AND NOT VLV07_ALMD_CNF_OPN_DN AND NOT VLV07_ALMD_CNF_CLS_DN AND %MW150:X0;

// Rung 208
  LD %M195                (* VLV07_ALMD_CNF_OPN_DN *)
  OR %M196                (* VLV07_ALMD_CNF_CLS_DN *)
  OR %M181                (* VLV07_HMI_STP *)
  ST %M191                (* VLV07_SAVE_DATETIME *)
  // as ST:
  //   VLV07_SAVE_DATETIME := VLV07_ALMD_CNF_OPN_DN OR VLV07_ALMD_CNF_CLS_DN OR VLV07_HMI_STP;

// Rung 209: MSJ
  LD 1
  [ %C34.P := %MW64 ]     (* VLV07_CNT_HR, VLV07_WORK_CICLE *)
  // as ST:
  //   VLV07_CNT_HR.P := VLV07_WORK_CICLE;

// Rung 210
  LD 1
  OPER [ %MW97 := %C33.V ](* VLV07_CNT_MIN *)
  [ %MW96 := %C34.V ]     (* VLV07_CNT_HR *)
  // as ST:
  //   %MW97 := VLV07_CNT_MIN.V;
  //   %MW96 := VLV07_CNT_HR.V;

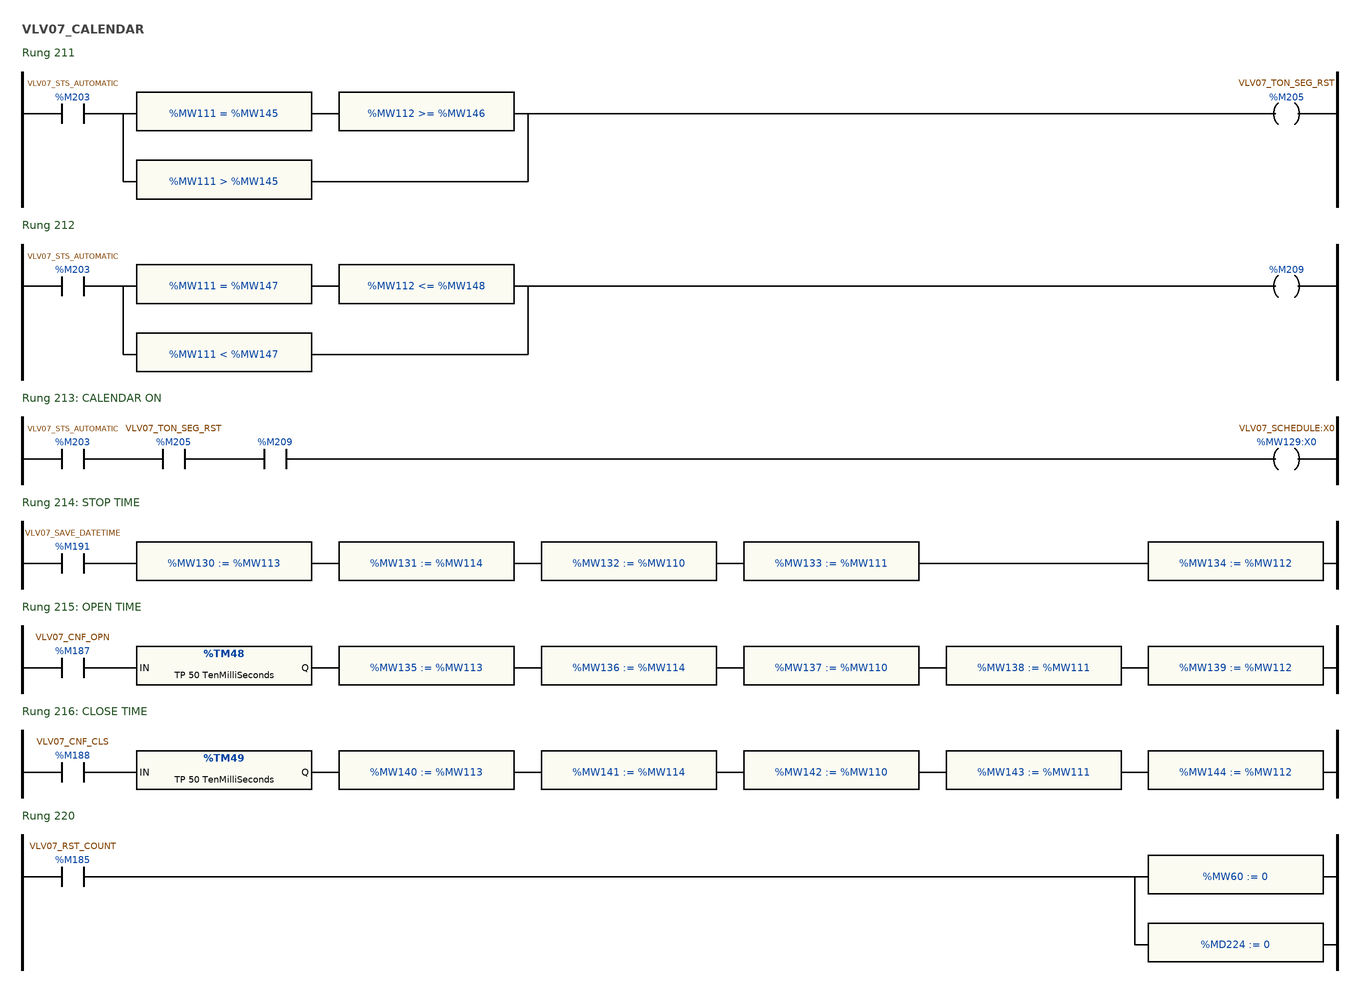

// Rung 211
  LD %M203                (* VLV07_STS_AUTOMATIC *)
  AND( [ %MW111 = %MW145 ](* HOUR, VLV07_SCHED_HR *)
  AND [ %MW112 >= %MW146 ](* MINUTES, VLV07_SCHED_MIN *)
  OR [ %MW111 > %MW145 ]  (* HOUR, VLV07_SCHED_HR *)
  )
  ST %M205                (* VLV07_TON_SEG_RST *)
  // as ST:
  //   VLV07_TON_SEG_RST := VLV07_STS_AUTOMATIC AND (HOUR = VLV07_SCHED_HR AND MINUTES >= VLV07_SCHED_MIN OR HOUR > VLV07_SCHED_HR);

// Rung 212
  LD %M203                (* VLV07_STS_AUTOMATIC *)
  AND( [ %MW111 = %MW147 ](* HOUR *)
  AND [ %MW112 <= %MW148 ](* MINUTES *)
  OR [ %MW111 < %MW147 ]  (* HOUR *)
  )
  ST %M209
  // as ST:
  //   %M209 := VLV07_STS_AUTOMATIC AND (HOUR = %MW147 AND MINUTES <= %MW148 OR HOUR < %MW147);

// Rung 213: CALENDAR ON
  LD %M203                (* VLV07_STS_AUTOMATIC *)
  AND %M205               (* VLV07_TON_SEG_RST *)
  AND %M209
  ST %MW129:X0            (* VLV07_SCHEDULE *)
  // as ST:
  //   VLV07_SCHEDULE:X0 := VLV07_STS_AUTOMATIC AND VLV07_TON_SEG_RST AND %M209;

// Rung 214: STOP TIME
  LD %M191                (* VLV07_SAVE_DATETIME *)
  OPER [ %MW130 := %MW113 ](* VLV07_MONTH, MONTH *)
  OPER [ %MW131 := %MW114 ](* VLV07_YR, YEAR *)
  OPER [ %MW132 := %MW110 ](* VLV07_DY, DAY *)
  OPER [ %MW133 := %MW111 ](* VLV07_HR, HOUR *)
  [ %MW134 := %MW112 ]    (* VLV07_MIN, MINUTES *)
  // as ST:
  //   IF VLV07_SAVE_DATETIME THEN VLV07_MONTH := MONTH; END_IF;
  //   IF VLV07_SAVE_DATETIME THEN VLV07_YR := YEAR; END_IF;
  //   IF VLV07_SAVE_DATETIME THEN VLV07_DY := DAY; END_IF;
  //   IF VLV07_SAVE_DATETIME THEN VLV07_HR := HOUR; END_IF;
  //   IF VLV07_SAVE_DATETIME THEN VLV07_MIN := MINUTES; END_IF;

// Rung 215: OPEN TIME
  BLK %TM48
  LD %M187                (* VLV07_CNF_OPN *)
  IN
  OUT_BLK
  LD Q
  OPER [ %MW135 := %MW113 ](* VLV07_OPEN_MONTH, MONTH *)
  OPER [ %MW136 := %MW114 ](* VLV07_OPEN_YR, YEAR *)
  OPER [ %MW137 := %MW110 ](* VLV07_OPEN_DY, DAY *)
  OPER [ %MW138 := %MW111 ](* VLV07_OPEN_HR, HOUR *)
  [ %MW139 := %MW112 ]    (* VLV07_OPEN_MIN, MINUTES *)
  END_BLK
  // as ST:
  //   %TM48(IN := VLV07_CNF_OPN);
  //   IF %TM48.Q THEN VLV07_OPEN_MONTH := MONTH; END_IF;
  //   IF %TM48.Q THEN VLV07_OPEN_YR := YEAR; END_IF;
  //   IF %TM48.Q THEN VLV07_OPEN_DY := DAY; END_IF;
  //   IF %TM48.Q THEN VLV07_OPEN_HR := HOUR; END_IF;
  //   IF %TM48.Q THEN VLV07_OPEN_MIN := MINUTES; END_IF;

// Rung 216: CLOSE TIME
  BLK %TM49
  LD %M188                (* VLV07_CNF_CLS *)
  IN
  OUT_BLK
  LD Q
  OPER [ %MW140 := %MW113 ](* VLV07_CLOSE_MONTH, MONTH *)
  OPER [ %MW141 := %MW114 ](* VLV07_CLOSE_YR, YEAR *)
  OPER [ %MW142 := %MW110 ](* VLV07_CLOSE_DY, DAY *)
  OPER [ %MW143 := %MW111 ](* VLV07_CLOSE_HR, HOUR *)
  [ %MW144 := %MW112 ]    (* VLV07_CLOSE_MIN, MINUTES *)
  END_BLK
  // as ST:
  //   %TM49(IN := VLV07_CNF_CLS);
  //   IF %TM49.Q THEN VLV07_CLOSE_MONTH := MONTH; END_IF;
  //   IF %TM49.Q THEN VLV07_CLOSE_YR := YEAR; END_IF;
  //   IF %TM49.Q THEN VLV07_CLOSE_DY := DAY; END_IF;
  //   IF %TM49.Q THEN VLV07_CLOSE_HR := HOUR; END_IF;
  //   IF %TM49.Q THEN VLV07_CLOSE_MIN := MINUTES; END_IF;

// Rung 217
  BLK %C34                (* VLV07_CNT_HR *)
  LD %M185                (* VLV07_RST_COUNT *)
  OR( %M21                (* HORARIOOFICINA_ACTIVE *)
  RISING32
  )
  R
  LD %M207                (* VLV07_TON_MIN_DN *)
  CU
  OUT_BLK
  LD D
  ST %M208                (* VLV07_TON_HR_DN *)
  END_BLK
  // as ST:
  //   VLV07_CNT_HR(RISING32 := HORARIOOFICINA_ACTIVE, R := VLV07_RST_COUNT OR HORARIOOFICINA_ACTIVE, CU := VLV07_TON_MIN_DN);
  //   VLV07_TON_HR_DN := VLV07_CNT_HR.D;
  (* the ladder stored for this rung does not match its IL; not drawn *)

// Rung 218
  BLK %C33                (* VLV07_CNT_MIN *)
  LD 1
  AND( %M185              (* VLV07_RST_COUNT *)
  OR %M207                (* VLV07_TON_MIN_DN *)
  )
  OR( %M21                (* HORARIOOFICINA_ACTIVE *)
  RISING33
  )
  R
  LD %M206                (* VLV07_TON_SEG_DN *)
  CU
  OUT_BLK
  LD D
  ST %M207                (* VLV07_TON_MIN_DN *)
  END_BLK
  // as ST:
  //   VLV07_CNT_MIN(RISING33 := HORARIOOFICINA_ACTIVE, R := VLV07_RST_COUNT OR VLV07_TON_MIN_DN OR HORARIOOFICINA_ACTIVE, CU := VLV07_TON_SEG_DN);
  //   VLV07_TON_MIN_DN := VLV07_CNT_MIN.D;
  (* the ladder stored for this rung does not match its IL; not drawn *)

// Rung 219
  LD 1
  MULTIFB
  LD 1
  ST %MW2509:X1
  BLK %TM61
  LD %MW2509:X1
  AND %M203               (* VLV07_STS_AUTOMATIC *)
  ANDN %M206              (* VLV07_TON_SEG_DN *)
  IN
  OUT_BLK
  LD Q
  ST %MW2509:X0
  END_BLK
  BLK %C32                (* VLV07_CNT_SEG *)
  LD %MW2509:X1
  AND( %M185              (* VLV07_RST_COUNT *)
  OR %M206                (* VLV07_TON_SEG_DN *)
  )
  R
  LD %MW2509:X0
  CU
  OUT_BLK
  LD D
  ST %M206                (* VLV07_TON_SEG_DN *)
  END_BLK
  MULTIFB
  // as ST:
  //   %MW2509:X1 := TRUE;
  //   %TM61(IN := %MW2509:X1 AND VLV07_STS_AUTOMATIC AND NOT VLV07_TON_SEG_DN);
  //   %MW2509:X0 := %TM61.Q;
  //   VLV07_CNT_SEG(R := %MW2509:X1 AND (VLV07_RST_COUNT OR VLV07_TON_SEG_DN), CU := %MW2509:X0);
  //   VLV07_TON_SEG_DN := VLV07_CNT_SEG.D;
  (* the ladder stored for this rung does not match its IL; not drawn *)

// Rung 220
  LD %M185                (* VLV07_RST_COUNT *)
  [ %MW60 := 0 ]          (* VLV07_CNT_OPN_ACC *)
  [ %MD224 := 0 ]         (* VLV07_CNT_OPN_ACC2 *)
  // as ST:
  //   IF VLV07_RST_COUNT THEN VLV07_CNT_OPN_ACC := 0; END_IF;
  //   IF VLV07_RST_COUNT THEN VLV07_CNT_OPN_ACC2 := 0; END_IF;

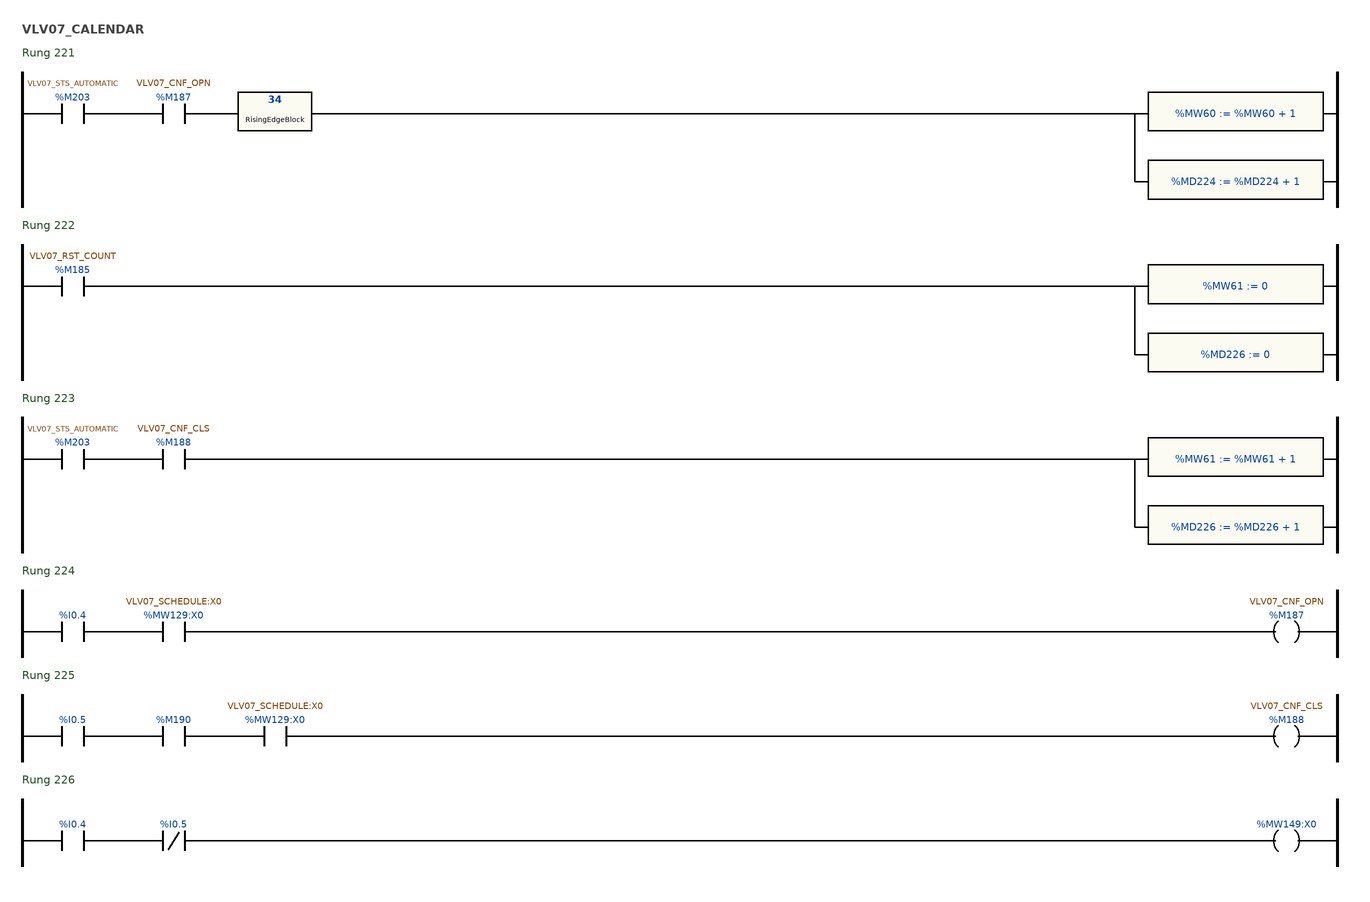

// Rung 221
  LD %M203                (* VLV07_STS_AUTOMATIC *)
  AND %M187               (* VLV07_CNF_OPN *)
  RISING34
  [ %MW60 := %MW60 + 1 ]  (* VLV07_CNT_OPN_ACC, VLV07_CNT_OPN_ACC *)
  [ %MD224 := %MD224 + 1 ](* VLV07_CNT_OPN_ACC2, VLV07_CNT_OPN_ACC2 *)
  // as ST:
  //   IF RISING(VLV07_STS_AUTOMATIC AND VLV07_CNF_OPN) THEN VLV07_CNT_OPN_ACC := VLV07_CNT_OPN_ACC + 1; END_IF;
  //   IF RISING(VLV07_STS_AUTOMATIC AND VLV07_CNF_OPN) THEN VLV07_CNT_OPN_ACC2 := VLV07_CNT_OPN_ACC2 + 1; END_IF;

// Rung 222
  LD %M185                (* VLV07_RST_COUNT *)
  [ %MW61 := 0 ]          (* VLV07_CNT_CLS_ACC *)
  [ %MD226 := 0 ]         (* VLV07_CNT_CLS_ACC2 *)
  // as ST:
  //   IF VLV07_RST_COUNT THEN VLV07_CNT_CLS_ACC := 0; END_IF;
  //   IF VLV07_RST_COUNT THEN VLV07_CNT_CLS_ACC2 := 0; END_IF;

// Rung 223
  LD %M203                (* VLV07_STS_AUTOMATIC *)
  AND %M188               (* VLV07_CNF_CLS *)
  [ %MW61 := %MW61 + 1 ]  (* VLV07_CNT_CLS_ACC, VLV07_CNT_CLS_ACC *)
  [ %MD226 := %MD226 + 1 ](* VLV07_CNT_CLS_ACC2, VLV07_CNT_CLS_ACC2 *)
  // as ST:
  //   IF VLV07_STS_AUTOMATIC AND VLV07_CNF_CLS THEN VLV07_CNT_CLS_ACC := VLV07_CNT_CLS_ACC + 1; END_IF;
  //   IF VLV07_STS_AUTOMATIC AND VLV07_CNF_CLS THEN VLV07_CNT_CLS_ACC2 := VLV07_CNT_CLS_ACC2 + 1; END_IF;

// Rung 224
  LD %I0.4
  AND %MW129:X0           (* VLV07_SCHEDULE *)
  ST %M187                (* VLV07_CNF_OPN *)
  // as ST:
  //   VLV07_CNF_OPN := %I0.4 AND VLV07_SCHEDULE:X0;

// Rung 225
  LD %I0.5
  AND %M190
  AND %MW129:X0           (* VLV07_SCHEDULE *)
  ST %M188                (* VLV07_CNF_CLS *)
  // as ST:
  //   VLV07_CNF_CLS := %I0.5 AND %M190 AND VLV07_SCHEDULE:X0;

// Rung 226
  LD %I0.4
  ANDN %I0.5
  ST %MW149:X0
  // as ST:
  //   %MW149:X0 := %I0.4 AND NOT %I0.5;

POU COMM
  (* SectionNumber=9 *)

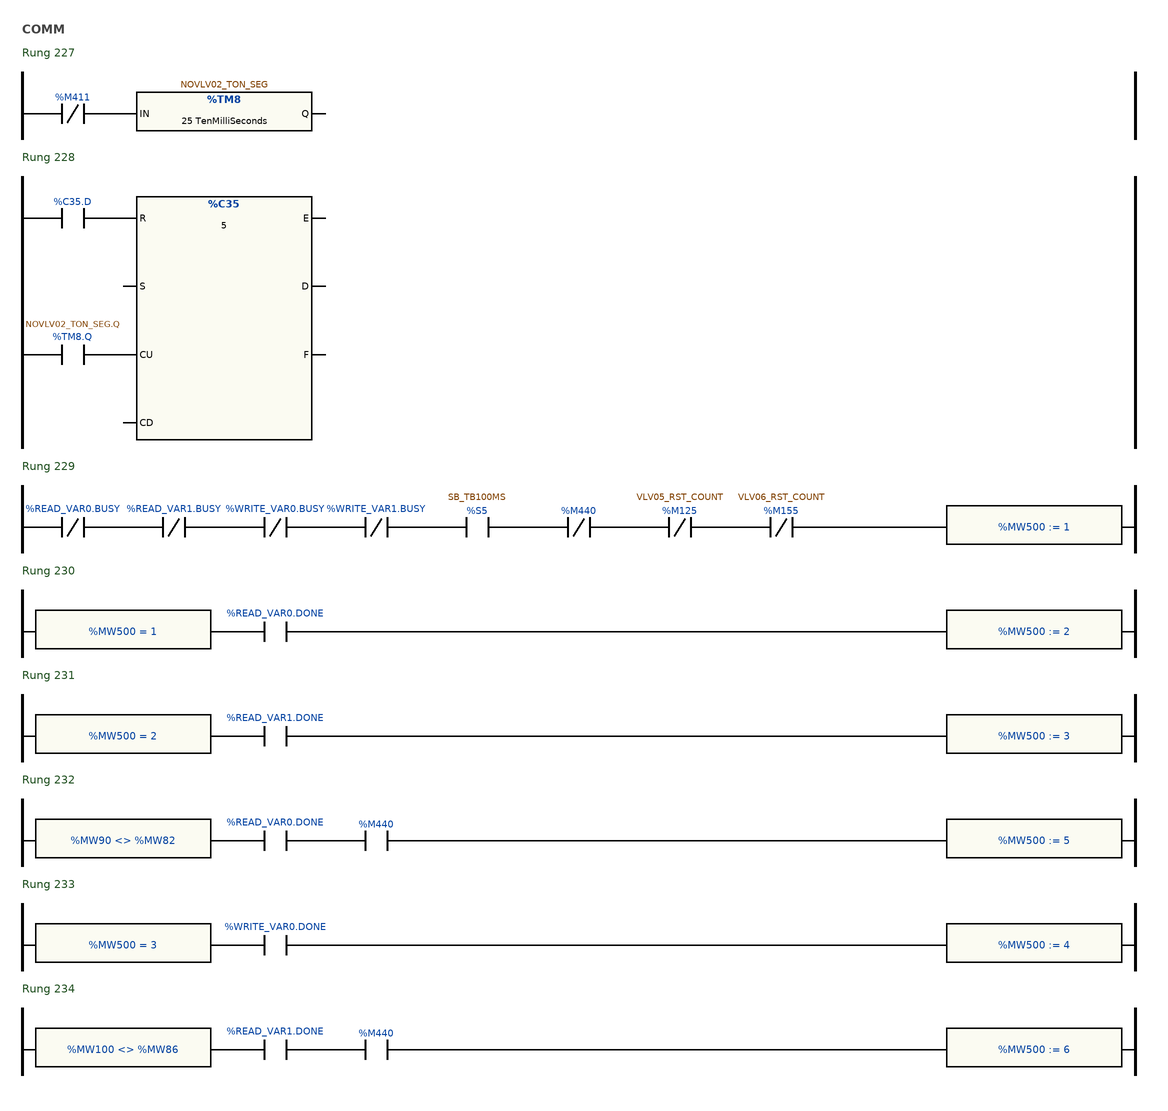

// Rung 227
  BLK %TM8                (* NOVLV02_TON_SEG *)
  LDN %M411
  IN
  END_BLK
  // as ST:
  //   NOVLV02_TON_SEG(IN := NOT %M411);

// Rung 228
  BLK %C35
  LD %C35.D
  R
  LD %TM8.Q               (* NOVLV02_TON_SEG *)
  CU
  END_BLK
  // as ST:
  //   %C35(R := %C35.D, CU := NOVLV02_TON_SEG.Q);

// Rung 229
  LDN %READ_VAR0.BUSY
  ANDN %READ_VAR1.BUSY
  ANDN %WRITE_VAR0.BUSY
  ANDN %WRITE_VAR1.BUSY
  AND %S5                 (* SB_TB100MS *)
  ANDN %M440
  ANDN %M125              (* VLV05_RST_COUNT *)
  ANDN %M155              (* VLV06_RST_COUNT *)
  [ %MW500 := 1 ]
  // as ST:
  //   IF NOT %READ_VAR0.BUSY AND NOT %READ_VAR1.BUSY AND NOT %WRITE_VAR0.BUSY AND NOT %WRITE_VAR1.BUSY AND SB_TB100MS AND NOT %M440 AND NOT VLV05_RST_COUNT AND NOT VLV06_RST_COUNT THEN %MW500 := 1; END_IF;

// Rung 230
  LD [ %MW500 = 1 ]
  AND %READ_VAR0.DONE
  [ %MW500 := 2 ]
  // as ST:
  //   IF %MW500 = 1 AND %READ_VAR0.DONE THEN %MW500 := 2; END_IF;

// Rung 231
  LD [ %MW500 = 2 ]
  AND %READ_VAR1.DONE
  [ %MW500 := 3 ]
  // as ST:
  //   IF %MW500 = 2 AND %READ_VAR1.DONE THEN %MW500 := 3; END_IF;

// Rung 232
  LD [ %MW90 <> %MW82 ]
  AND %READ_VAR0.DONE
  AND %M440
  [ %MW500 := 5 ]
  // as ST:
  //   IF %MW90 <> %MW82 AND %READ_VAR0.DONE AND %M440 THEN %MW500 := 5; END_IF;

// Rung 233
  LD [ %MW500 = 3 ]
  AND %WRITE_VAR0.DONE
  [ %MW500 := 4 ]
  // as ST:
  //   IF %MW500 = 3 AND %WRITE_VAR0.DONE THEN %MW500 := 4; END_IF;

// Rung 234
  LD [ %MW100 <> %MW86 ]
  AND %READ_VAR1.DONE
  AND %M440
  [ %MW500 := 6 ]
  // as ST:
  //   IF %MW100 <> %MW86 AND %READ_VAR1.DONE AND %M440 THEN %MW500 := 6; END_IF;

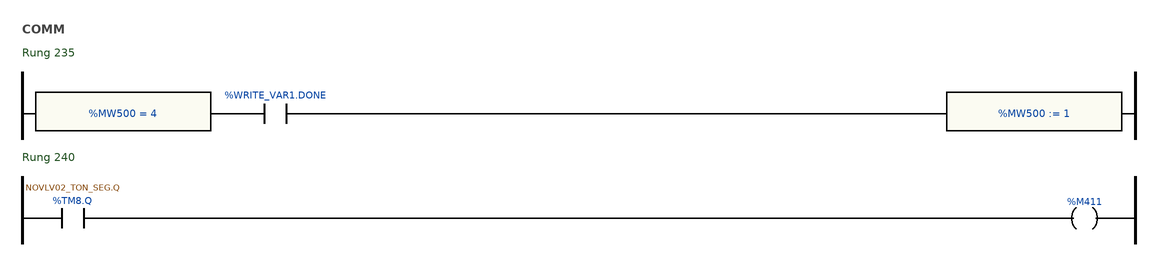

// Rung 235
  LD [ %MW500 = 4 ]
  AND %WRITE_VAR1.DONE
  [ %MW500 := 1 ]
  // as ST:
  //   IF %MW500 = 4 AND %WRITE_VAR1.DONE THEN %MW500 := 1; END_IF;

// Rung 236: R1
  BLK %READ_VAR0
  LD [ %C35.V = 0 ]
  RISING35
  EXECUTE
  LD [ %C35.V = 1 ]
  RISING36
  ABORT
  OUT_BLK
  LD DONE
  ST %M400
  LD BUSY
  ST %M402
  LD ABORTED
  ST %M403
  LD ERROR
  ST %M401
  END_BLK
  // as ST:
  //   %READ_VAR0(RISING35 := %C35.V = 0, EXECUTE := %C35.V = 0, RISING36 := %C35.V = 1, ABORT := %C35.V = 1);
  //   %M400 := %READ_VAR0.DONE;
  //   %M402 := %READ_VAR0.BUSY;
  //   %M403 := %READ_VAR0.ABORTED;
  //   %M401 := %READ_VAR0.ERROR;
  (* the ladder stored for this rung does not match its IL; not drawn *)

// Rung 237: W1
  BLK %WRITE_VAR0
  LD [ %C35.V = 1 ]
  RISING37
  EXECUTE
  LD [ %C35.V = 2 ]
  RISING38
  ABORT
  OUT_BLK
  LD DONE
  ST %M404
  LD BUSY
  ST %M405
  LD ABORTED
  ST %M406
  LD ERROR
  ST %M407
  END_BLK
  // as ST:
  //   %WRITE_VAR0(RISING37 := %C35.V = 1, EXECUTE := %C35.V = 1, RISING38 := %C35.V = 2, ABORT := %C35.V = 2);
  //   %M404 := %WRITE_VAR0.DONE;
  //   %M405 := %WRITE_VAR0.BUSY;
  //   %M406 := %WRITE_VAR0.ABORTED;
  //   %M407 := %WRITE_VAR0.ERROR;
  (* the ladder stored for this rung does not match its IL; not drawn *)

// Rung 238: R2
  BLK %READ_VAR1
  LD [ %C35.V = 2 ]
  RISING39
  EXECUTE
  LD [ %C35.V = 3 ]
  RISING40
  ABORT
  END_BLK
  // as ST:
  //   %READ_VAR1(RISING39 := %C35.V = 2, EXECUTE := %C35.V = 2, RISING40 := %C35.V = 3, ABORT := %C35.V = 3);
  (* the ladder stored for this rung does not match its IL; not drawn *)

// Rung 239: W2
  BLK %WRITE_VAR1
  LD [ %C35.V = 3 ]
  RISING41
  EXECUTE
  LD [ %C35.V = 4 ]
  RISING42
  ABORT
  END_BLK
  // as ST:
  //   %WRITE_VAR1(RISING41 := %C35.V = 3, EXECUTE := %C35.V = 3, RISING42 := %C35.V = 4, ABORT := %C35.V = 4);
  (* the ladder stored for this rung does not match its IL; not drawn *)

// Rung 240
  LD %TM8.Q               (* NOVLV02_TON_SEG *)
  ST %M411
  // as ST:
  //   %M411 := NOVLV02_TON_SEG.Q;

POU VLV08_MODBUS_CURRENT
  (* SectionNumber=10 *)

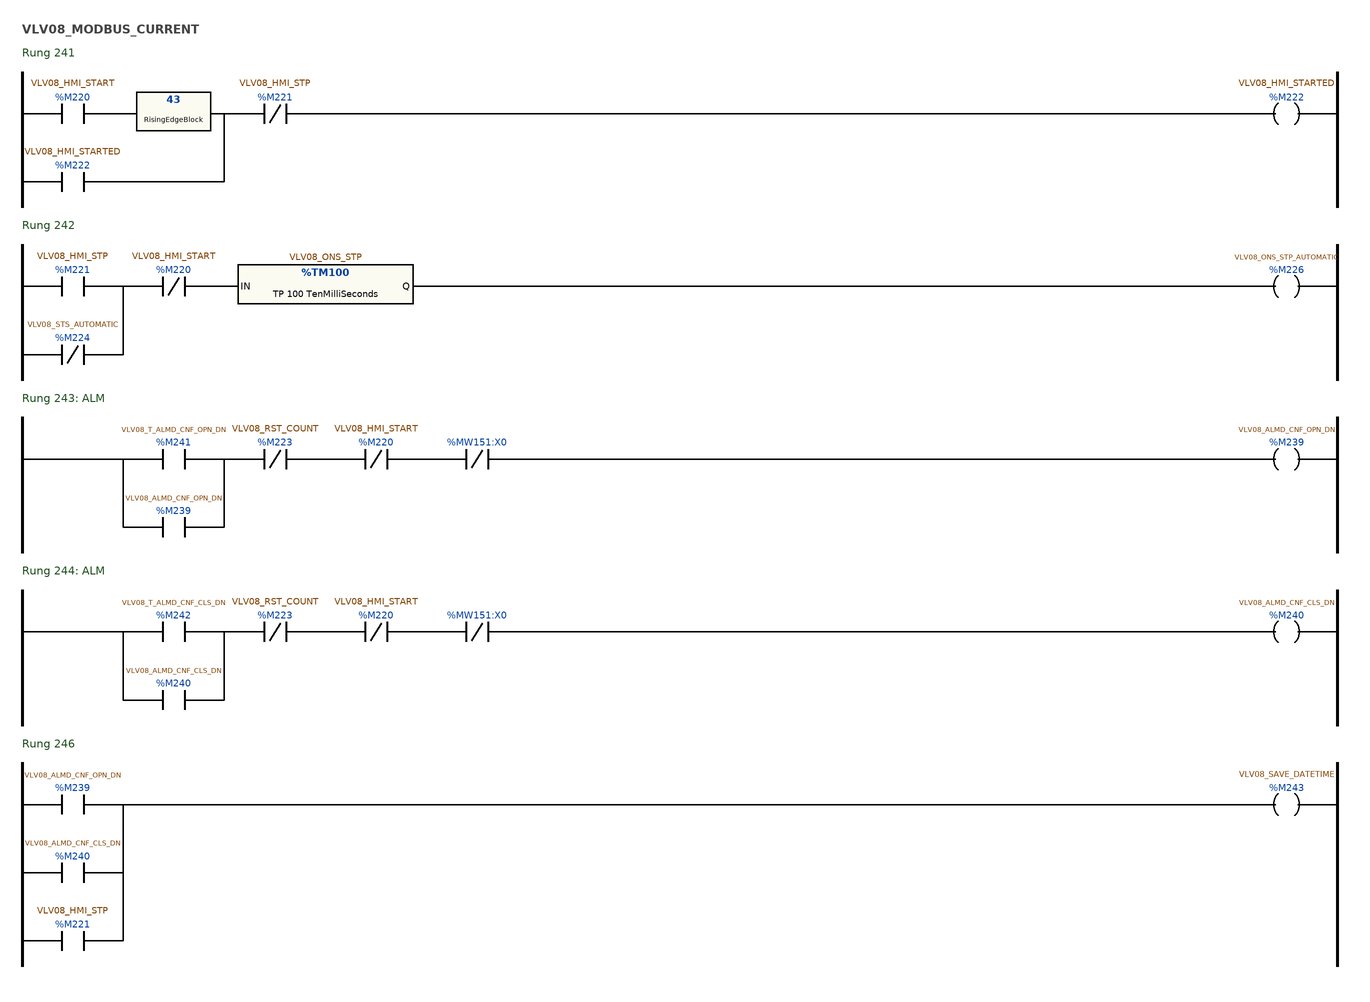

// Rung 241
  LD %M220                (* VLV08_HMI_START *)
  RISING43
  OR %M222                (* VLV08_HMI_STARTED *)
  ANDN %M221              (* VLV08_HMI_STP *)
  ST %M222                (* VLV08_HMI_STARTED *)
  // as ST:
  //   VLV08_HMI_STARTED := (RISING(VLV08_HMI_START) OR VLV08_HMI_STARTED) AND NOT VLV08_HMI_STP;

// Rung 242
  BLK %TM100              (* VLV08_ONS_STP *)
  LD %M221                (* VLV08_HMI_STP *)
  ORN %M224               (* VLV08_STS_AUTOMATIC *)
  ANDN %M220              (* VLV08_HMI_START *)
  IN
  OUT_BLK
  LD Q
  ST %M226                (* VLV08_ONS_STP_AUTOMATIC *)
  END_BLK
  // as ST:
  //   VLV08_ONS_STP(IN := (VLV08_HMI_STP OR NOT VLV08_STS_AUTOMATIC) AND NOT VLV08_HMI_START);
  //   VLV08_ONS_STP_AUTOMATIC := VLV08_ONS_STP.Q;

// Rung 243: ALM
  LD 1
  AND( %M241              (* VLV08_T_ALMD_CNF_OPN_DN *)
  OR %M239                (* VLV08_ALMD_CNF_OPN_DN *)
  )
  ANDN %M223              (* VLV08_RST_COUNT *)
  ANDN %M220              (* VLV08_HMI_START *)
  ANDN %MW151:X0
  ST %M239                (* VLV08_ALMD_CNF_OPN_DN *)
  // as ST:
  //   VLV08_ALMD_CNF_OPN_DN := (VLV08_T_ALMD_CNF_OPN_DN OR VLV08_ALMD_CNF_OPN_DN) AND NOT VLV08_RST_COUNT AND NOT VLV08_HMI_START AND NOT %MW151:X0;

// Rung 244: ALM
  LD 1
  AND( %M242              (* VLV08_T_ALMD_CNF_CLS_DN *)
  OR %M240                (* VLV08_ALMD_CNF_CLS_DN *)
  )
  ANDN %M223              (* VLV08_RST_COUNT *)
  ANDN %M220              (* VLV08_HMI_START *)
  ANDN %MW151:X0
  ST %M240                (* VLV08_ALMD_CNF_CLS_DN *)
  // as ST:
  //   VLV08_ALMD_CNF_CLS_DN := (VLV08_T_ALMD_CNF_CLS_DN OR VLV08_ALMD_CNF_CLS_DN) AND NOT VLV08_RST_COUNT AND NOT VLV08_HMI_START AND NOT %MW151:X0;

// Rung 245
  LD 1
  MULTIFB
  LD 1
  AND %M21                (* HORARIOOFICINA_ACTIVE *)
  AND %M222               (* VLV08_HMI_STARTED *)
  ANDN %M239              (* VLV08_ALMD_CNF_OPN_DN *)
  ANDN %M240              (* VLV08_ALMD_CNF_CLS_DN *)
  AND %MW432:X0
  ANDN %M238              (* VLV08_TON_HR_DN *)
  ST %MW2509:X0
  LD %MW2509:X0
  ST %M224                (* VLV08_STS_AUTOMATIC *)
  BLK %TM101              (* VLV08_ONS_02 *)
  LD %MW2509:X0
  IN
  OUT_BLK
  LD Q
  ST %M250                (* VLV08_ONS_STR_AUTOMATIC *)
  END_BLK
  MULTIFB
  // as ST:
  //   %MW2509:X0 := HORARIOOFICINA_ACTIVE AND VLV08_HMI_STARTED AND NOT VLV08_ALMD_CNF_OPN_DN AND NOT VLV08_ALMD_CNF_CLS_DN AND %MW432:X0 AND NOT VLV08_TON_HR_DN;
  //   VLV08_STS_AUTOMATIC := %MW2509:X0;
  //   VLV08_ONS_02(IN := %MW2509:X0);
  //   VLV08_ONS_STR_AUTOMATIC := VLV08_ONS_02.Q;
  (* the ladder stored for this rung does not match its IL; not drawn *)

// Rung 246
  LD %M239                (* VLV08_ALMD_CNF_OPN_DN *)
  OR %M240                (* VLV08_ALMD_CNF_CLS_DN *)
  OR %M221                (* VLV08_HMI_STP *)
  ST %M243                (* VLV08_SAVE_DATETIME *)
  // as ST:
  //   VLV08_SAVE_DATETIME := VLV08_ALMD_CNF_OPN_DN OR VLV08_ALMD_CNF_CLS_DN OR VLV08_HMI_STP;

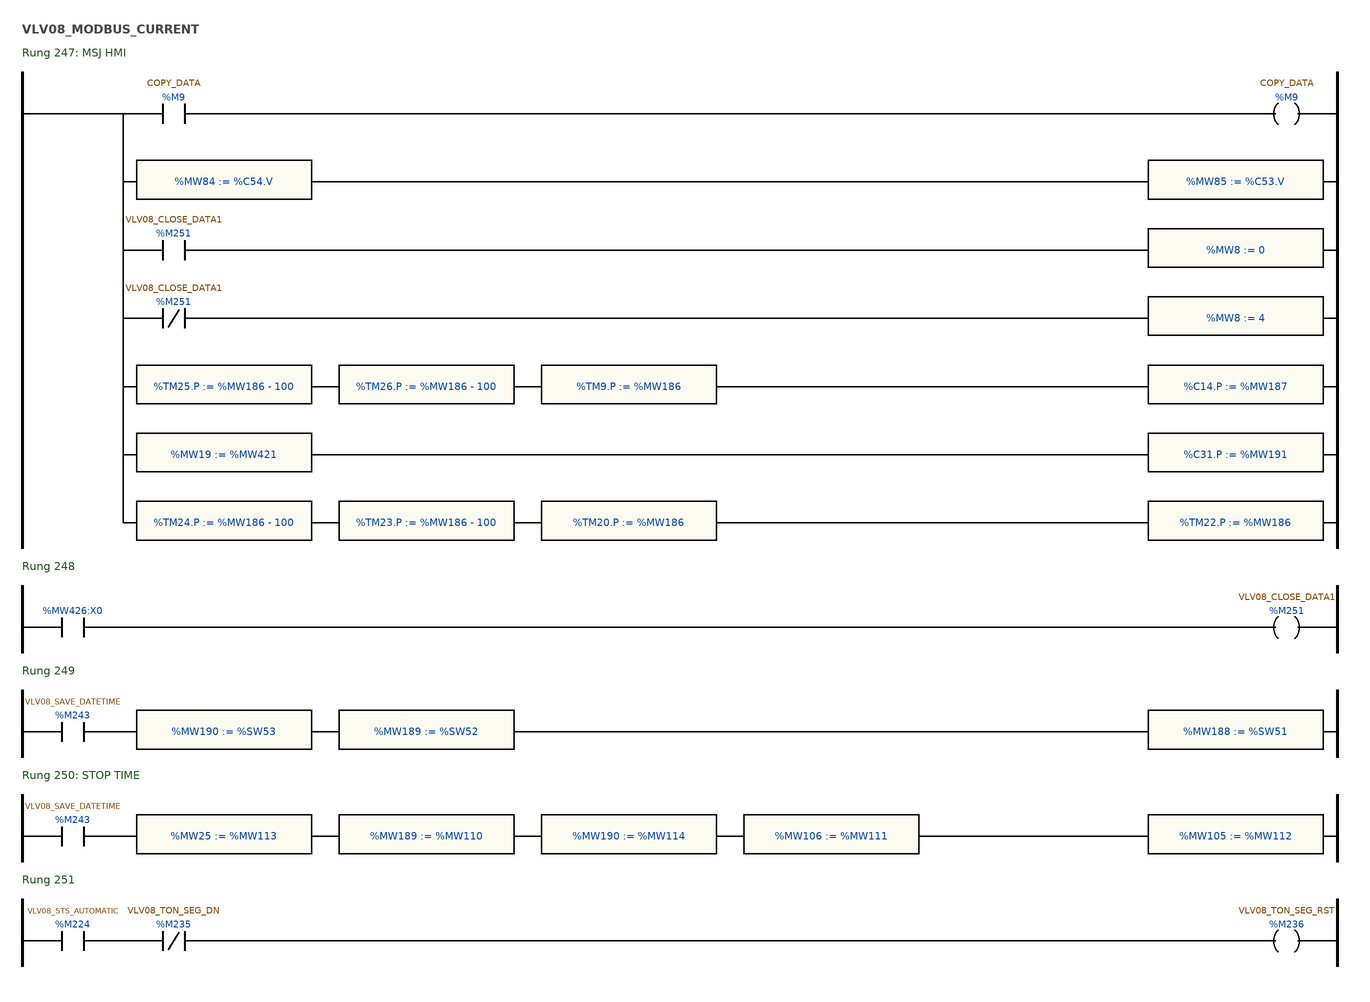

// Rung 247: MSJ HMI
  LD 1
  MPS
  AND %M9                 (* COPY_DATA *)
  ST %M9                  (* COPY_DATA *)
  MRD
  OPER [ %MW84 := %C54.V ](* VLV08_CNT_HR *)
  [ %MW85 := %C53.V ]     (* VLV08_CNT_MIN *)
  MRD
  AND %M251               (* VLV08_CLOSE_DATA1 *)
  [ %MW8 := 0 ]
  MRD
  ANDN %M251              (* VLV08_CLOSE_DATA1 *)
  [ %MW8 := 4 ]
  MRD
  OPER [ %TM25.P := %MW186 - 100 ](* VLV03_T_CNF_OPN, VLV08_T_CNF_PRESET *)
  OPER [ %TM26.P := %MW186 - 100 ](* VLV03_T_CNF_CLS, VLV08_T_CNF_PRESET *)
  OPER [ %TM9.P := %MW186 ](* VLV03_ONS_STP, VLV08_T_CNF_PRESET *)
  [ %C14.P := %MW187 ]    (* VLV03_CNT_HR, VLV08_CNF_HR_PRESET *)
  MRD
  OPER [ %MW19 := %MW421 ](* VLV03_CV_ACTUAL *)
  [ %C31.P := %MW191 ]    (* VLV08_SETPOINT_ALTO *)
  MPP
  OPER [ %TM24.P := %MW186 - 100 ](* VLV03_TON_ALMD_CNF_CLS, VLV08_T_CNF_PRESET *)
  OPER [ %TM23.P := %MW186 - 100 ](* VLV03_TON_ALMD_CNF_OPN, VLV08_T_CNF_PRESET *)
  OPER [ %TM20.P := %MW186 ](* VLV03_TON_OPN, VLV08_T_CNF_PRESET *)
  [ %TM22.P := %MW186 ]   (* VLV03_TON_CLS, VLV08_T_CNF_PRESET *)
  // as ST:
  //   COPY_DATA := COPY_DATA;
  //   %MW84 := VLV08_CNT_HR.V;
  //   %MW85 := VLV08_CNT_MIN.V;
  //   IF VLV08_CLOSE_DATA1 THEN %MW8 := 0; END_IF;
  //   IF NOT VLV08_CLOSE_DATA1 THEN %MW8 := 4; END_IF;
  //   VLV03_T_CNF_OPN.P := VLV08_T_CNF_PRESET - 100;
  //   VLV03_T_CNF_CLS.P := VLV08_T_CNF_PRESET - 100;
  //   VLV03_ONS_STP.P := VLV08_T_CNF_PRESET;
  //   VLV03_CNT_HR.P := VLV08_CNF_HR_PRESET;
  //   VLV03_CV_ACTUAL := %MW421;
  //   %C31.P := VLV08_SETPOINT_ALTO;
  //   VLV03_TON_ALMD_CNF_CLS.P := VLV08_T_CNF_PRESET - 100;
  //   VLV03_TON_ALMD_CNF_OPN.P := VLV08_T_CNF_PRESET - 100;
  //   VLV03_TON_OPN.P := VLV08_T_CNF_PRESET;
  //   VLV03_TON_CLS.P := VLV08_T_CNF_PRESET;

// Rung 248
  (* no IL stored for this rung *)

// Rung 249
  LD %M243                (* VLV08_SAVE_DATETIME *)
  OPER [ %MW190 := %SW53 ](* VLV08_RTC_YY, SW_RTCCCYY *)
  OPER [ %MW189 := %SW52 ](* VLV08_RTC_MMDD, SW_RTCMMDD *)
  [ %MW188 := %SW51 ]     (* VLV08_RTC_HHMM, SW_RTCHHMM *)
  // as ST:
  //   IF VLV08_SAVE_DATETIME THEN VLV08_RTC_YY := SW_RTCCCYY; END_IF;
  //   IF VLV08_SAVE_DATETIME THEN VLV08_RTC_MMDD := SW_RTCMMDD; END_IF;
  //   IF VLV08_SAVE_DATETIME THEN VLV08_RTC_HHMM := SW_RTCHHMM; END_IF;

// Rung 250: STOP TIME
  LD %M243                (* VLV08_SAVE_DATETIME *)
  OPER [ %MW25 := %MW113 ](* VLV03_RTC_HHMM, MONTH *)
  OPER [ %MW189 := %MW110 ](* VLV08_RTC_MMDD, DAY *)
  OPER [ %MW190 := %MW114 ](* VLV08_RTC_YY, YEAR *)
  OPER [ %MW106 := %MW111 ](* HOUR *)
  [ %MW105 := %MW112 ]    (* MINUTES *)
  // as ST:
  //   IF VLV08_SAVE_DATETIME THEN VLV03_RTC_HHMM := MONTH; END_IF;
  //   IF VLV08_SAVE_DATETIME THEN VLV08_RTC_MMDD := DAY; END_IF;
  //   IF VLV08_SAVE_DATETIME THEN VLV08_RTC_YY := YEAR; END_IF;
  //   IF VLV08_SAVE_DATETIME THEN %MW106 := HOUR; END_IF;
  //   IF VLV08_SAVE_DATETIME THEN %MW105 := MINUTES; END_IF;

// Rung 251
  LD %M224                (* VLV08_STS_AUTOMATIC *)
  ANDN %M235              (* VLV08_TON_SEG_DN *)
  ST %M236                (* VLV08_TON_SEG_RST *)
  // as ST:
  //   VLV08_TON_SEG_RST := VLV08_STS_AUTOMATIC AND NOT VLV08_TON_SEG_DN;

// Rung 252
  BLK %C14                (* VLV03_CNT_HR *)
  LD %M223                (* VLV08_RST_COUNT *)
  OR( %M21                (* HORARIOOFICINA_ACTIVE *)
  RISING53
  )
  R
  LD %M237                (* VLV08_TON_MIN_DN *)
  CU
  OUT_BLK
  LD D
  ST %M238                (* VLV08_TON_HR_DN *)
  END_BLK
  // as ST:
  //   VLV03_CNT_HR(RISING53 := HORARIOOFICINA_ACTIVE, R := VLV08_RST_COUNT OR HORARIOOFICINA_ACTIVE, CU := VLV08_TON_MIN_DN);
  //   VLV08_TON_HR_DN := VLV03_CNT_HR.D;
  (* the ladder stored for this rung does not match its IL; not drawn *)

// Rung 253
  BLK %C13                (* VLV03_CNT_MIN *)
  LD 1
  AND( %M223              (* VLV08_RST_COUNT *)
  OR %M237                (* VLV08_TON_MIN_DN *)
  )
  OR( %M21                (* HORARIOOFICINA_ACTIVE *)
  RISING53
  )
  R
  LD %M235                (* VLV08_TON_SEG_DN *)
  CU
  OUT_BLK
  LD D
  ST %M237                (* VLV08_TON_MIN_DN *)
  END_BLK
  // as ST:
  //   VLV03_CNT_MIN(RISING53 := HORARIOOFICINA_ACTIVE, R := VLV08_RST_COUNT OR VLV08_TON_MIN_DN OR HORARIOOFICINA_ACTIVE, CU := VLV08_TON_SEG_DN);
  //   VLV08_TON_MIN_DN := VLV03_CNT_MIN.D;
  (* the ladder stored for this rung does not match its IL; not drawn *)

// Rung 254
  LD 1
  MULTIFB
  LD 1
  ST %MW2509:X1
  BLK %TM21               (* VLV03_TON_SEG *)
  LD %MW2509:X1
  AND %M224               (* VLV08_STS_AUTOMATIC *)
  AND %M236               (* VLV08_TON_SEG_RST *)
  IN
  OUT_BLK
  LD Q
  ST %MW2509:X0
  END_BLK
  BLK %C12                (* VLV03_CNT_SEG *)
  LD %MW2509:X1
  AND( %M223              (* VLV08_RST_COUNT *)
  OR %M235                (* VLV08_TON_SEG_DN *)
  )
  R
  LD %MW2509:X0
  CU
  OUT_BLK
  LD D
  ST %M235                (* VLV08_TON_SEG_DN *)
  END_BLK
  MULTIFB
  // as ST:
  //   %MW2509:X1 := TRUE;
  //   VLV03_TON_SEG(IN := %MW2509:X1 AND VLV08_STS_AUTOMATIC AND VLV08_TON_SEG_RST);
  //   %MW2509:X0 := VLV03_TON_SEG.Q;
  //   VLV03_CNT_SEG(R := %MW2509:X1 AND (VLV08_RST_COUNT OR VLV08_TON_SEG_DN), CU := %MW2509:X0);
  //   VLV08_TON_SEG_DN := VLV03_CNT_SEG.D;
  (* the ladder stored for this rung does not match its IL; not drawn *)

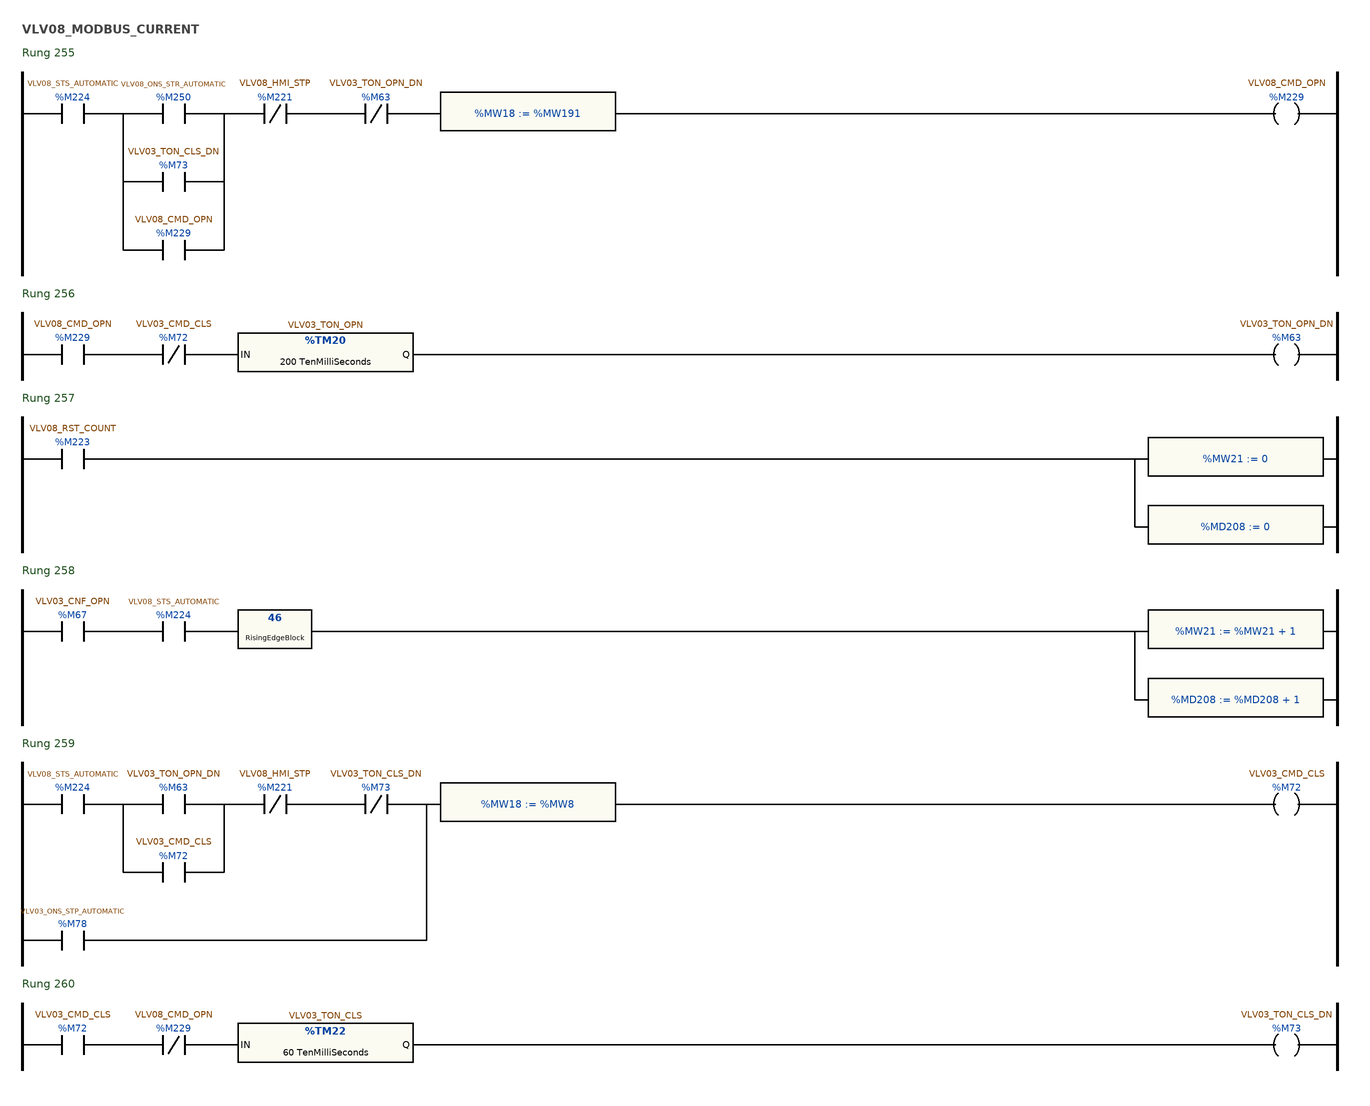

// Rung 255
  LD %M224                (* VLV08_STS_AUTOMATIC *)
  AND( %M250              (* VLV08_ONS_STR_AUTOMATIC *)
  OR %M73                 (* VLV03_TON_CLS_DN *)
  OR %M229                (* VLV08_CMD_OPN *)
  )
  ANDN %M221              (* VLV08_HMI_STP *)
  ANDN %M63               (* VLV03_TON_OPN_DN *)
  OPER [ %MW18 := %MW191 ](* VLV03_SP_ACTUAL, VLV08_SETPOINT_ALTO *)
  ST %M229                (* VLV08_CMD_OPN *)
  // as ST:
  //   IF VLV08_STS_AUTOMATIC AND (VLV08_ONS_STR_AUTOMATIC OR VLV03_TON_CLS_DN OR VLV08_CMD_OPN) AND NOT VLV08_HMI_STP AND NOT VLV03_TON_OPN_DN THEN VLV03_SP_ACTUAL := VLV08_SETPOINT_ALTO; END_IF;
  //   VLV08_CMD_OPN := VLV08_STS_AUTOMATIC AND (VLV08_ONS_STR_AUTOMATIC OR VLV03_TON_CLS_DN OR VLV08_CMD_OPN) AND NOT VLV08_HMI_STP AND NOT VLV03_TON_OPN_DN;

// Rung 256
  BLK %TM20               (* VLV03_TON_OPN *)
  LD %M229                (* VLV08_CMD_OPN *)
  ANDN %M72               (* VLV03_CMD_CLS *)
  IN
  OUT_BLK
  LD Q
  ST %M63                 (* VLV03_TON_OPN_DN *)
  END_BLK
  // as ST:
  //   VLV03_TON_OPN(IN := VLV08_CMD_OPN AND NOT VLV03_CMD_CLS);
  //   VLV03_TON_OPN_DN := VLV03_TON_OPN.Q;

// Rung 257
  LD %M223                (* VLV08_RST_COUNT *)
  [ %MW21 := 0 ]          (* VLV03_CNT_OPN_ACC *)
  [ %MD208 := 0 ]         (* VLV03_CNT_OPN_ACC2 *)
  // as ST:
  //   IF VLV08_RST_COUNT THEN VLV03_CNT_OPN_ACC := 0; END_IF;
  //   IF VLV08_RST_COUNT THEN VLV03_CNT_OPN_ACC2 := 0; END_IF;

// Rung 258
  LD %M67                 (* VLV03_CNF_OPN *)
  AND %M224               (* VLV08_STS_AUTOMATIC *)
  RISING46
  [ %MW21 := %MW21 + 1 ]  (* VLV03_CNT_OPN_ACC, VLV03_CNT_OPN_ACC *)
  [ %MD208 := %MD208 + 1 ](* VLV03_CNT_OPN_ACC2, VLV03_CNT_OPN_ACC2 *)
  // as ST:
  //   IF RISING(VLV03_CNF_OPN AND VLV08_STS_AUTOMATIC) THEN VLV03_CNT_OPN_ACC := VLV03_CNT_OPN_ACC + 1; END_IF;
  //   IF RISING(VLV03_CNF_OPN AND VLV08_STS_AUTOMATIC) THEN VLV03_CNT_OPN_ACC2 := VLV03_CNT_OPN_ACC2 + 1; END_IF;

// Rung 259
  LD %M224                (* VLV08_STS_AUTOMATIC *)
  AND( %M63               (* VLV03_TON_OPN_DN *)
  OR %M72                 (* VLV03_CMD_CLS *)
  )
  ANDN %M221              (* VLV08_HMI_STP *)
  ANDN %M73               (* VLV03_TON_CLS_DN *)
  OR %M78                 (* VLV03_ONS_STP_AUTOMATIC *)
  OPER [ %MW18 := %MW8 ]  (* VLV03_SP_ACTUAL *)
  ST %M72                 (* VLV03_CMD_CLS *)
  // as ST:
  //   IF VLV08_STS_AUTOMATIC AND (VLV03_TON_OPN_DN OR VLV03_CMD_CLS) AND NOT VLV08_HMI_STP AND NOT VLV03_TON_CLS_DN OR VLV03_ONS_STP_AUTOMATIC THEN VLV03_SP_ACTUAL := %MW8; END_IF;
  //   VLV03_CMD_CLS := VLV08_STS_AUTOMATIC AND (VLV03_TON_OPN_DN OR VLV03_CMD_CLS) AND NOT VLV08_HMI_STP AND NOT VLV03_TON_CLS_DN OR VLV03_ONS_STP_AUTOMATIC;

// Rung 260
  BLK %TM22               (* VLV03_TON_CLS *)
  LD %M72                 (* VLV03_CMD_CLS *)
  ANDN %M229              (* VLV08_CMD_OPN *)
  IN
  OUT_BLK
  LD Q
  ST %M73                 (* VLV03_TON_CLS_DN *)
  END_BLK
  // as ST:
  //   VLV03_TON_CLS(IN := VLV03_CMD_CLS AND NOT VLV08_CMD_OPN);
  //   VLV03_TON_CLS_DN := VLV03_TON_CLS.Q;

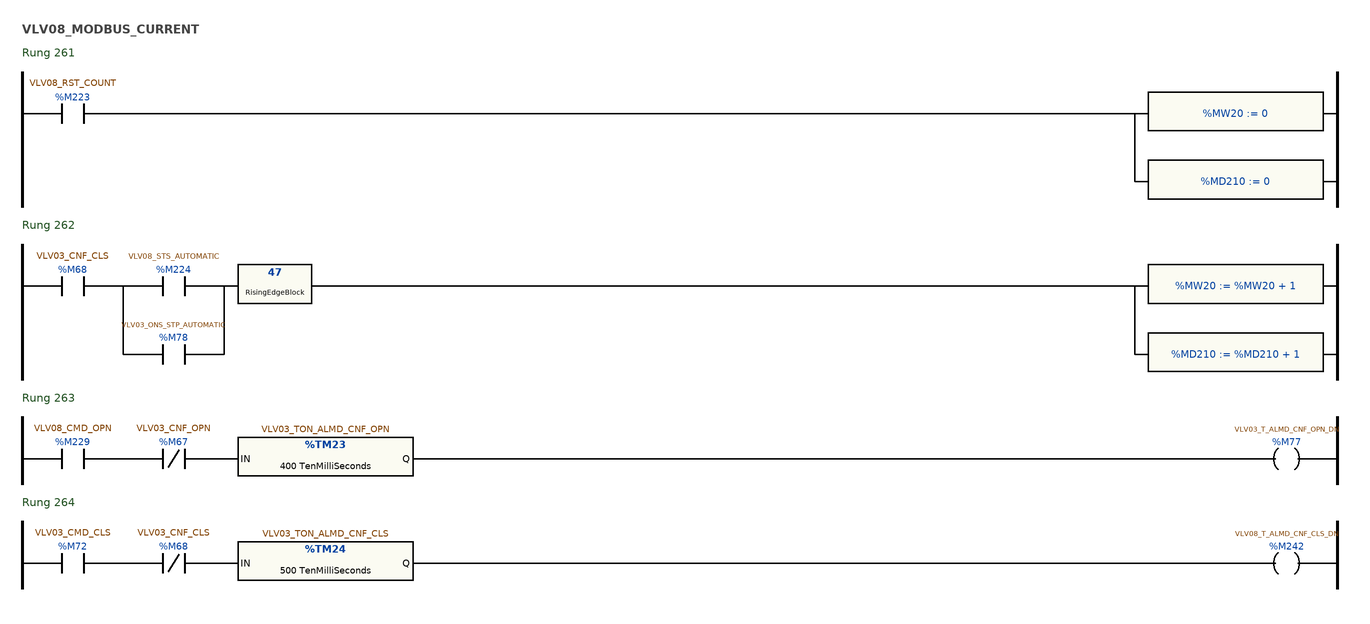

// Rung 261
  LD %M223                (* VLV08_RST_COUNT *)
  [ %MW20 := 0 ]          (* VLV03_CNT_CLS_ACC *)
  [ %MD210 := 0 ]         (* VLV03_CNT_CLS_ACC2 *)
  // as ST:
  //   IF VLV08_RST_COUNT THEN VLV03_CNT_CLS_ACC := 0; END_IF;
  //   IF VLV08_RST_COUNT THEN VLV03_CNT_CLS_ACC2 := 0; END_IF;

// Rung 262
  LD %M68                 (* VLV03_CNF_CLS *)
  AND( %M224              (* VLV08_STS_AUTOMATIC *)
  OR %M78                 (* VLV03_ONS_STP_AUTOMATIC *)
  )
  RISING47
  [ %MW20 := %MW20 + 1 ]  (* VLV03_CNT_CLS_ACC, VLV03_CNT_CLS_ACC *)
  [ %MD210 := %MD210 + 1 ](* VLV03_CNT_CLS_ACC2, VLV03_CNT_CLS_ACC2 *)
  // as ST:
  //   IF RISING(VLV03_CNF_CLS AND (VLV08_STS_AUTOMATIC OR VLV03_ONS_STP_AUTOMATIC)) THEN VLV03_CNT_CLS_ACC := VLV03_CNT_CLS_ACC + 1; END_IF;
  //   IF RISING(VLV03_CNF_CLS AND (VLV08_STS_AUTOMATIC OR VLV03_ONS_STP_AUTOMATIC)) THEN VLV03_CNT_CLS_ACC2 := VLV03_CNT_CLS_ACC2 + 1; END_IF;

// Rung 263
  BLK %TM23               (* VLV03_TON_ALMD_CNF_OPN *)
  LD %M229                (* VLV08_CMD_OPN *)
  ANDN %M67               (* VLV03_CNF_OPN *)
  IN
  OUT_BLK
  LD Q
  ST %M77                 (* VLV03_T_ALMD_CNF_OPN_DN *)
  END_BLK
  // as ST:
  //   VLV03_TON_ALMD_CNF_OPN(IN := VLV08_CMD_OPN AND NOT VLV03_CNF_OPN);
  //   VLV03_T_ALMD_CNF_OPN_DN := VLV03_TON_ALMD_CNF_OPN.Q;

// Rung 264
  BLK %TM24               (* VLV03_TON_ALMD_CNF_CLS *)
  LD %M72                 (* VLV03_CMD_CLS *)
  ANDN %M68               (* VLV03_CNF_CLS *)
  IN
  OUT_BLK
  LD Q
  ST %M242                (* VLV08_T_ALMD_CNF_CLS_DN *)
  END_BLK
  // as ST:
  //   VLV03_TON_ALMD_CNF_CLS(IN := VLV03_CMD_CLS AND NOT VLV03_CNF_CLS);
  //   VLV08_T_ALMD_CNF_CLS_DN := VLV03_TON_ALMD_CNF_CLS.Q;

POU VLV09_MODBUS_VOLTAGE
  (* SectionNumber=11 *)

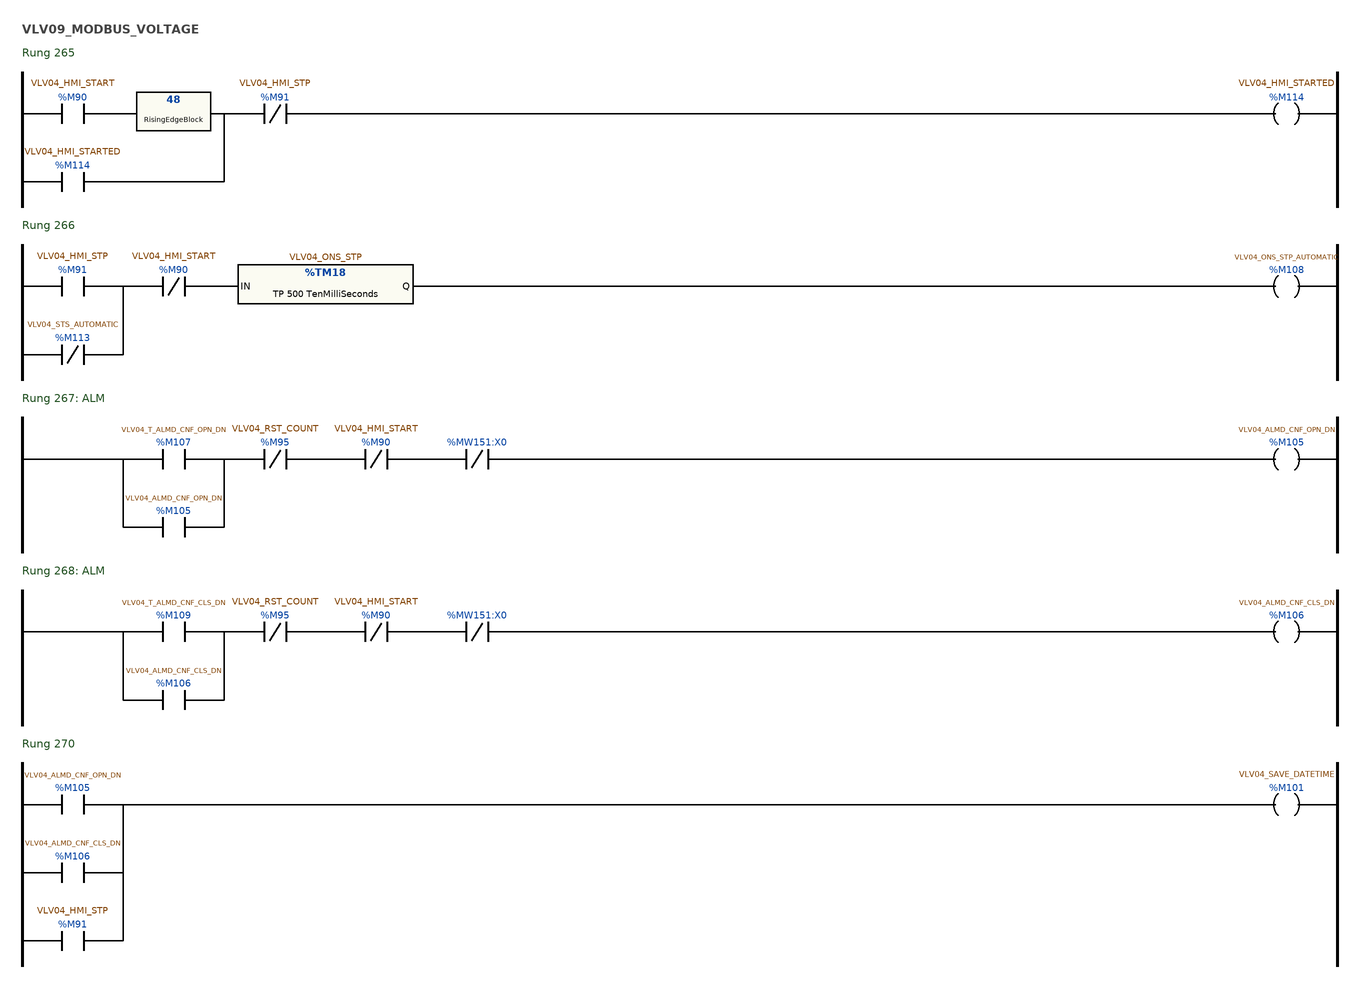

// Rung 265
  LD %M90                 (* VLV04_HMI_START *)
  RISING48
  OR %M114                (* VLV04_HMI_STARTED *)
  ANDN %M91               (* VLV04_HMI_STP *)
  ST %M114                (* VLV04_HMI_STARTED *)
  // as ST:
  //   VLV04_HMI_STARTED := (RISING(VLV04_HMI_START) OR VLV04_HMI_STARTED) AND NOT VLV04_HMI_STP;

// Rung 266
  BLK %TM18               (* VLV04_ONS_STP *)
  LD %M91                 (* VLV04_HMI_STP *)
  ORN %M113               (* VLV04_STS_AUTOMATIC *)
  ANDN %M90               (* VLV04_HMI_START *)
  IN
  OUT_BLK
  LD Q
  ST %M108                (* VLV04_ONS_STP_AUTOMATIC *)
  END_BLK
  // as ST:
  //   VLV04_ONS_STP(IN := (VLV04_HMI_STP OR NOT VLV04_STS_AUTOMATIC) AND NOT VLV04_HMI_START);
  //   VLV04_ONS_STP_AUTOMATIC := VLV04_ONS_STP.Q;

// Rung 267: ALM
  LD 1
  AND( %M107              (* VLV04_T_ALMD_CNF_OPN_DN *)
  OR %M105                (* VLV04_ALMD_CNF_OPN_DN *)
  )
  ANDN %M95               (* VLV04_RST_COUNT *)
  ANDN %M90               (* VLV04_HMI_START *)
  ANDN %MW151:X0
  ST %M105                (* VLV04_ALMD_CNF_OPN_DN *)
  // as ST:
  //   VLV04_ALMD_CNF_OPN_DN := (VLV04_T_ALMD_CNF_OPN_DN OR VLV04_ALMD_CNF_OPN_DN) AND NOT VLV04_RST_COUNT AND NOT VLV04_HMI_START AND NOT %MW151:X0;

// Rung 268: ALM
  LD 1
  AND( %M109              (* VLV04_T_ALMD_CNF_CLS_DN *)
  OR %M106                (* VLV04_ALMD_CNF_CLS_DN *)
  )
  ANDN %M95               (* VLV04_RST_COUNT *)
  ANDN %M90               (* VLV04_HMI_START *)
  ANDN %MW151:X0
  ST %M106                (* VLV04_ALMD_CNF_CLS_DN *)
  // as ST:
  //   VLV04_ALMD_CNF_CLS_DN := (VLV04_T_ALMD_CNF_CLS_DN OR VLV04_ALMD_CNF_CLS_DN) AND NOT VLV04_RST_COUNT AND NOT VLV04_HMI_START AND NOT %MW151:X0;

// Rung 269
  LD 1
  MULTIFB
  LD 1
  AND %M21                (* HORARIOOFICINA_ACTIVE *)
  AND %M114               (* VLV04_HMI_STARTED *)
  ANDN %M105              (* VLV04_ALMD_CNF_OPN_DN *)
  ANDN %M106              (* VLV04_ALMD_CNF_CLS_DN *)
  AND %MW432:X0
  ANDN %M118              (* VLV04_TON_HR_DN *)
  ST %MW2509:X0
  LD %MW2509:X0
  ST %M113                (* VLV04_STS_AUTOMATIC *)
  BLK %TM37               (* VLV04_ONS *)
  LD %MW2509:X0
  IN
  OUT_BLK
  LD Q
  ST %M96                 (* VLV04_ONS_STR_AUTOMATIC *)
  END_BLK
  MULTIFB
  // as ST:
  //   %MW2509:X0 := HORARIOOFICINA_ACTIVE AND VLV04_HMI_STARTED AND NOT VLV04_ALMD_CNF_OPN_DN AND NOT VLV04_ALMD_CNF_CLS_DN AND %MW432:X0 AND NOT VLV04_TON_HR_DN;
  //   VLV04_STS_AUTOMATIC := %MW2509:X0;
  //   VLV04_ONS(IN := %MW2509:X0);
  //   VLV04_ONS_STR_AUTOMATIC := VLV04_ONS.Q;
  (* the ladder stored for this rung does not match its IL; not drawn *)

// Rung 270
  LD %M105                (* VLV04_ALMD_CNF_OPN_DN *)
  OR %M106                (* VLV04_ALMD_CNF_CLS_DN *)
  OR %M91                 (* VLV04_HMI_STP *)
  ST %M101                (* VLV04_SAVE_DATETIME *)
  // as ST:
  //   VLV04_SAVE_DATETIME := VLV04_ALMD_CNF_OPN_DN OR VLV04_ALMD_CNF_CLS_DN OR VLV04_HMI_STP;

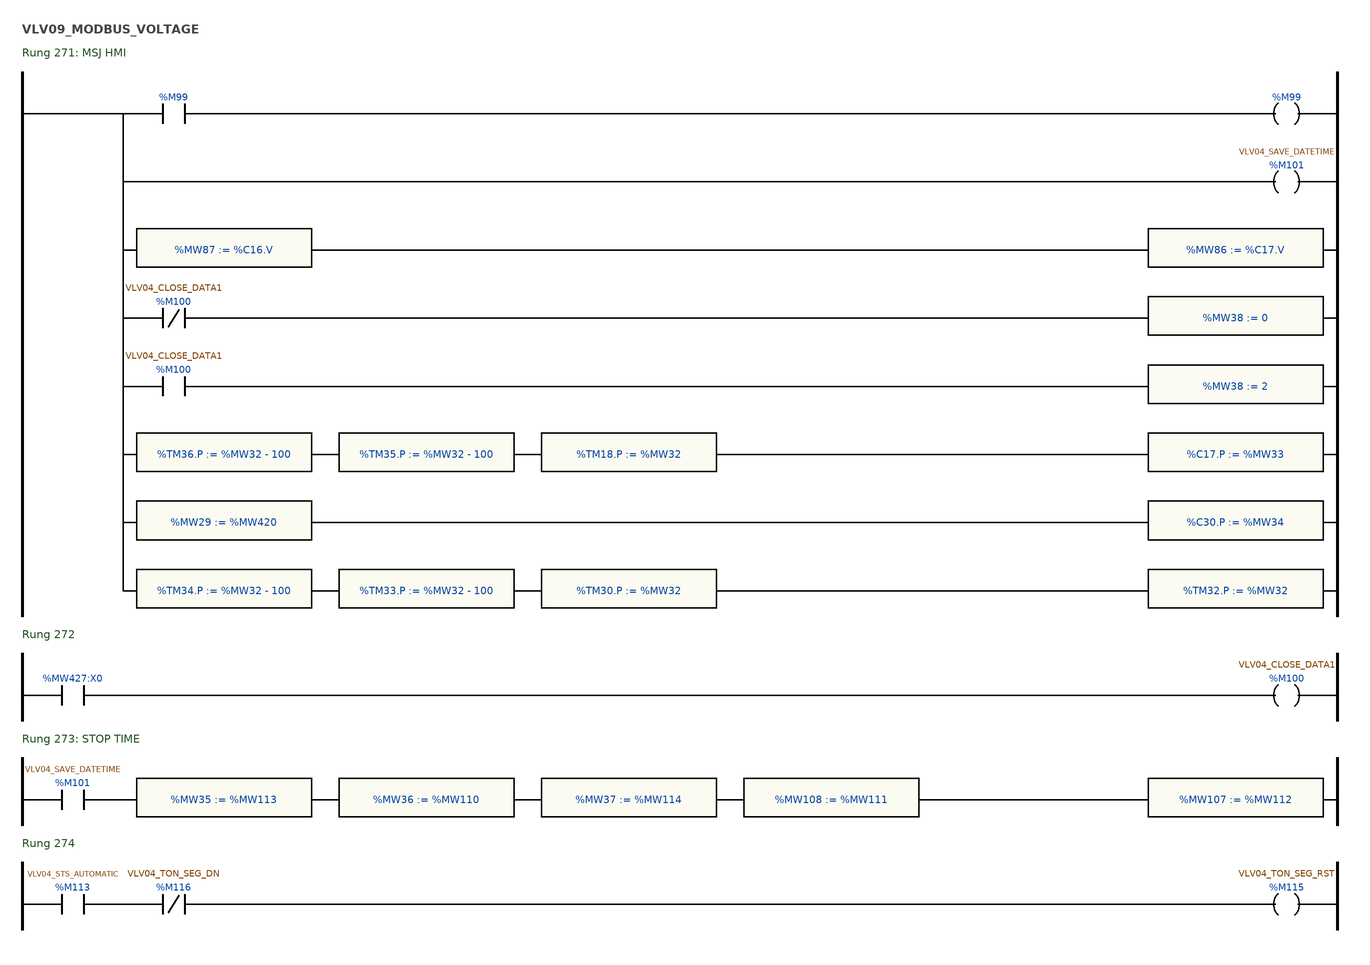

// Rung 271: MSJ HMI
  LD 1
  MPS
  AND %M99
  ST %M99
  MRD
  ST %M101                (* VLV04_SAVE_DATETIME *)
  MRD
  OPER [ %MW87 := %C16.V ](* VLV04_CNT_MIN *)
  [ %MW86 := %C17.V ]     (* VLV04_CNT_HR *)
  MRD
  ANDN %M100              (* VLV04_CLOSE_DATA1 *)
  [ %MW38 := 0 ]
  MRD
  AND %M100               (* VLV04_CLOSE_DATA1 *)
  [ %MW38 := 2 ]
  MRD
  OPER [ %TM36.P := %MW32 - 100 ](* VLV04_T_CNF_CLS, VLV04_T_CNF_PRESET *)
  OPER [ %TM35.P := %MW32 - 100 ](* VLV04_T_CNF_OPN, VLV04_T_CNF_PRESET *)
  OPER [ %TM18.P := %MW32 ](* VLV04_ONS_STP, VLV04_T_CNF_PRESET *)
  [ %C17.P := %MW33 ]     (* VLV04_CNT_HR, VLV04_CNF_HR_PRESET *)
  MRD
  OPER [ %MW29 := %MW420 ](* VLV04_CV_ACTUAL *)
  [ %C30.P := %MW34 ]     (* VLV04_SETPOINT_ALTO *)
  MPP
  OPER [ %TM34.P := %MW32 - 100 ](* VLV04_TON_ALMD_CNF_CLS, VLV04_T_CNF_PRESET *)
  OPER [ %TM33.P := %MW32 - 100 ](* VLV04_TON_ALMD_CNF_OPN, VLV04_T_CNF_PRESET *)
  OPER [ %TM30.P := %MW32 ](* VLV04_TON_OPN, VLV04_T_CNF_PRESET *)
  [ %TM32.P := %MW32 ]    (* VLV04_TON_CLS, VLV04_T_CNF_PRESET *)
  // as ST:
  //   %M99 := %M99;
  //   VLV04_SAVE_DATETIME := TRUE;
  //   %MW87 := VLV04_CNT_MIN.V;
  //   %MW86 := VLV04_CNT_HR.V;
  //   IF NOT VLV04_CLOSE_DATA1 THEN %MW38 := 0; END_IF;
  //   IF VLV04_CLOSE_DATA1 THEN %MW38 := 2; END_IF;
  //   VLV04_T_CNF_CLS.P := VLV04_T_CNF_PRESET - 100;
  //   VLV04_T_CNF_OPN.P := VLV04_T_CNF_PRESET - 100;
  //   VLV04_ONS_STP.P := VLV04_T_CNF_PRESET;
  //   VLV04_CNT_HR.P := VLV04_CNF_HR_PRESET;
  //   VLV04_CV_ACTUAL := %MW420;
  //   %C30.P := VLV04_SETPOINT_ALTO;
  //   VLV04_TON_ALMD_CNF_CLS.P := VLV04_T_CNF_PRESET - 100;
  //   VLV04_TON_ALMD_CNF_OPN.P := VLV04_T_CNF_PRESET - 100;
  //   VLV04_TON_OPN.P := VLV04_T_CNF_PRESET;
  //   VLV04_TON_CLS.P := VLV04_T_CNF_PRESET;

// Rung 272
  LD %MW427:X0
  ST %M100                (* VLV04_CLOSE_DATA1 *)
  // as ST:
  //   VLV04_CLOSE_DATA1 := %MW427:X0;

// Rung 273: STOP TIME
  LD %M101                (* VLV04_SAVE_DATETIME *)
  OPER [ %MW35 := %MW113 ](* VLV04_RTC_HHMM, MONTH *)
  OPER [ %MW36 := %MW110 ](* VLV04_RTC_MMDD, DAY *)
  OPER [ %MW37 := %MW114 ](* VLV04_RTC_YY, YEAR *)
  OPER [ %MW108 := %MW111 ](* HOUR *)
  [ %MW107 := %MW112 ]    (* MINUTES *)
  // as ST:
  //   IF VLV04_SAVE_DATETIME THEN VLV04_RTC_HHMM := MONTH; END_IF;
  //   IF VLV04_SAVE_DATETIME THEN VLV04_RTC_MMDD := DAY; END_IF;
  //   IF VLV04_SAVE_DATETIME THEN VLV04_RTC_YY := YEAR; END_IF;
  //   IF VLV04_SAVE_DATETIME THEN %MW108 := HOUR; END_IF;
  //   IF VLV04_SAVE_DATETIME THEN %MW107 := MINUTES; END_IF;

// Rung 274
  LD %M113                (* VLV04_STS_AUTOMATIC *)
  ANDN %M116              (* VLV04_TON_SEG_DN *)
  ST %M115                (* VLV04_TON_SEG_RST *)
  // as ST:
  //   VLV04_TON_SEG_RST := VLV04_STS_AUTOMATIC AND NOT VLV04_TON_SEG_DN;

// Rung 275
  BLK %C17                (* VLV04_CNT_HR *)
  LD %M95                 (* VLV04_RST_COUNT *)
  OR( %M21                (* HORARIOOFICINA_ACTIVE *)
  RISING49
  )
  R
  LD %M117                (* VLV04_TON_MIN_DN *)
  CU
  OUT_BLK
  LD D
  ST %M118                (* VLV04_TON_HR_DN *)
  END_BLK
  // as ST:
  //   VLV04_CNT_HR(RISING49 := HORARIOOFICINA_ACTIVE, R := VLV04_RST_COUNT OR HORARIOOFICINA_ACTIVE, CU := VLV04_TON_MIN_DN);
  //   VLV04_TON_HR_DN := VLV04_CNT_HR.D;
  (* the ladder stored for this rung does not match its IL; not drawn *)

// Rung 276
  BLK %C16                (* VLV04_CNT_MIN *)
  LD 1
  AND( %M95               (* VLV04_RST_COUNT *)
  OR %M117                (* VLV04_TON_MIN_DN *)
  )
  OR( %M21                (* HORARIOOFICINA_ACTIVE *)
  RISING50
  )
  R
  LD %M116                (* VLV04_TON_SEG_DN *)
  CU
  OUT_BLK
  LD D
  ST %M117                (* VLV04_TON_MIN_DN *)
  END_BLK
  // as ST:
  //   VLV04_CNT_MIN(RISING50 := HORARIOOFICINA_ACTIVE, R := VLV04_RST_COUNT OR VLV04_TON_MIN_DN OR HORARIOOFICINA_ACTIVE, CU := VLV04_TON_SEG_DN);
  //   VLV04_TON_MIN_DN := VLV04_CNT_MIN.D;
  (* the ladder stored for this rung does not match its IL; not drawn *)

// Rung 277
  LD 1
  MULTIFB
  LD 1
  ST %MW2509:X1
  BLK %TM31               (* VLV04_TON_SEG *)
  LD %MW2509:X1
  AND %M113               (* VLV04_STS_AUTOMATIC *)
  AND %M115               (* VLV04_TON_SEG_RST *)
  IN
  OUT_BLK
  LD Q
  ST %MW2509:X0
  END_BLK
  BLK %C15                (* VLV04_CNT_SEG *)
  LD %MW2509:X1
  AND( %M95               (* VLV04_RST_COUNT *)
  OR %M116                (* VLV04_TON_SEG_DN *)
  )
  R
  LD %MW2509:X0
  CU
  OUT_BLK
  LD D
  ST %M116                (* VLV04_TON_SEG_DN *)
  END_BLK
  MULTIFB
  // as ST:
  //   %MW2509:X1 := TRUE;
  //   VLV04_TON_SEG(IN := %MW2509:X1 AND VLV04_STS_AUTOMATIC AND VLV04_TON_SEG_RST);
  //   %MW2509:X0 := VLV04_TON_SEG.Q;
  //   VLV04_CNT_SEG(R := %MW2509:X1 AND (VLV04_RST_COUNT OR VLV04_TON_SEG_DN), CU := %MW2509:X0);
  //   VLV04_TON_SEG_DN := VLV04_CNT_SEG.D;
  (* the ladder stored for this rung does not match its IL; not drawn *)

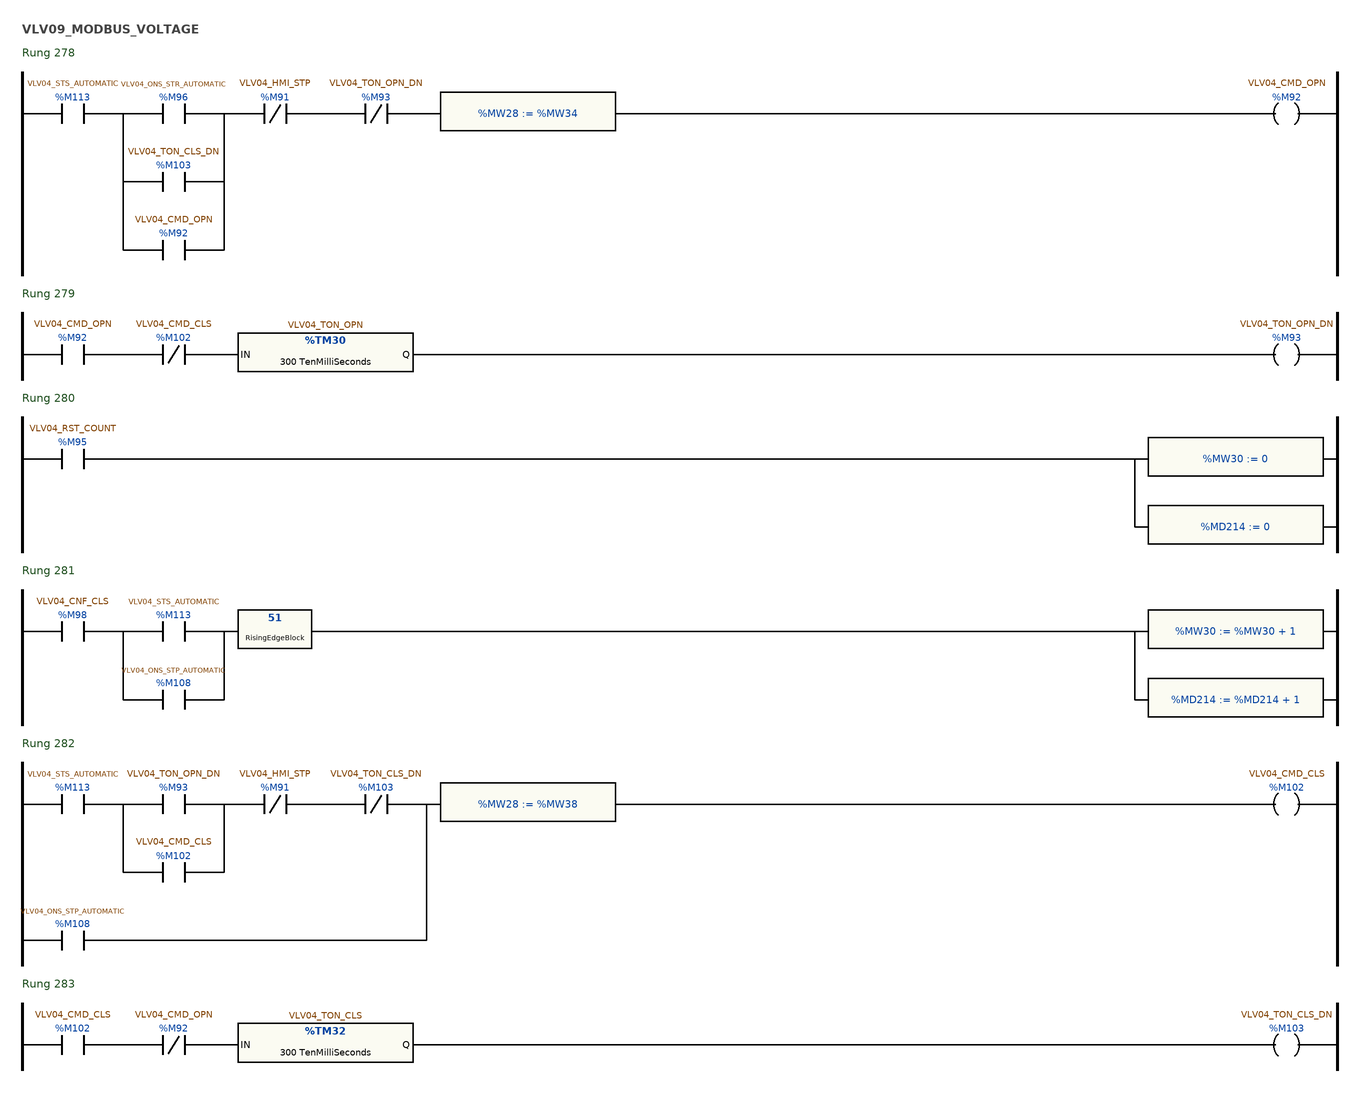

// Rung 278
  LD %M113                (* VLV04_STS_AUTOMATIC *)
  AND( %M96               (* VLV04_ONS_STR_AUTOMATIC *)
  OR %M103                (* VLV04_TON_CLS_DN *)
  OR %M92                 (* VLV04_CMD_OPN *)
  )
  ANDN %M91               (* VLV04_HMI_STP *)
  ANDN %M93               (* VLV04_TON_OPN_DN *)
  OPER [ %MW28 := %MW34 ] (* VLV04_SP_ACTUAL, VLV04_SETPOINT_ALTO *)
  ST %M92                 (* VLV04_CMD_OPN *)
  // as ST:
  //   IF VLV04_STS_AUTOMATIC AND (VLV04_ONS_STR_AUTOMATIC OR VLV04_TON_CLS_DN OR VLV04_CMD_OPN) AND NOT VLV04_HMI_STP AND NOT VLV04_TON_OPN_DN THEN VLV04_SP_ACTUAL := VLV04_SETPOINT_ALTO; END_IF;
  //   VLV04_CMD_OPN := VLV04_STS_AUTOMATIC AND (VLV04_ONS_STR_AUTOMATIC OR VLV04_TON_CLS_DN OR VLV04_CMD_OPN) AND NOT VLV04_HMI_STP AND NOT VLV04_TON_OPN_DN;

// Rung 279
  BLK %TM30               (* VLV04_TON_OPN *)
  LD %M92                 (* VLV04_CMD_OPN *)
  ANDN %M102              (* VLV04_CMD_CLS *)
  IN
  OUT_BLK
  LD Q
  ST %M93                 (* VLV04_TON_OPN_DN *)
  END_BLK
  // as ST:
  //   VLV04_TON_OPN(IN := VLV04_CMD_OPN AND NOT VLV04_CMD_CLS);
  //   VLV04_TON_OPN_DN := VLV04_TON_OPN.Q;

// Rung 280
  LD %M95                 (* VLV04_RST_COUNT *)
  [ %MW30 := 0 ]          (* VLV04_CNT_CLS_ACC *)
  [ %MD214 := 0 ]         (* VLV04_CNT_CLS_ACC2 *)
  // as ST:
  //   IF VLV04_RST_COUNT THEN VLV04_CNT_CLS_ACC := 0; END_IF;
  //   IF VLV04_RST_COUNT THEN VLV04_CNT_CLS_ACC2 := 0; END_IF;

// Rung 281
  LD %M98                 (* VLV04_CNF_CLS *)
  AND( %M113              (* VLV04_STS_AUTOMATIC *)
  OR %M108                (* VLV04_ONS_STP_AUTOMATIC *)
  )
  RISING51
  [ %MW30 := %MW30 + 1 ]  (* VLV04_CNT_CLS_ACC, VLV04_CNT_CLS_ACC *)
  [ %MD214 := %MD214 + 1 ](* VLV04_CNT_CLS_ACC2, VLV04_CNT_CLS_ACC2 *)
  // as ST:
  //   IF RISING(VLV04_CNF_CLS AND (VLV04_STS_AUTOMATIC OR VLV04_ONS_STP_AUTOMATIC)) THEN VLV04_CNT_CLS_ACC := VLV04_CNT_CLS_ACC + 1; END_IF;
  //   IF RISING(VLV04_CNF_CLS AND (VLV04_STS_AUTOMATIC OR VLV04_ONS_STP_AUTOMATIC)) THEN VLV04_CNT_CLS_ACC2 := VLV04_CNT_CLS_ACC2 + 1; END_IF;

// Rung 282
  LD %M113                (* VLV04_STS_AUTOMATIC *)
  AND( %M93               (* VLV04_TON_OPN_DN *)
  OR %M102                (* VLV04_CMD_CLS *)
  )
  ANDN %M91               (* VLV04_HMI_STP *)
  ANDN %M103              (* VLV04_TON_CLS_DN *)
  OR %M108                (* VLV04_ONS_STP_AUTOMATIC *)
  OPER [ %MW28 := %MW38 ] (* VLV04_SP_ACTUAL *)
  ST %M102                (* VLV04_CMD_CLS *)
  // as ST:
  //   IF VLV04_STS_AUTOMATIC AND (VLV04_TON_OPN_DN OR VLV04_CMD_CLS) AND NOT VLV04_HMI_STP AND NOT VLV04_TON_CLS_DN OR VLV04_ONS_STP_AUTOMATIC THEN VLV04_SP_ACTUAL := %MW38; END_IF;
  //   VLV04_CMD_CLS := VLV04_STS_AUTOMATIC AND (VLV04_TON_OPN_DN OR VLV04_CMD_CLS) AND NOT VLV04_HMI_STP AND NOT VLV04_TON_CLS_DN OR VLV04_ONS_STP_AUTOMATIC;

// Rung 283
  BLK %TM32               (* VLV04_TON_CLS *)
  LD %M102                (* VLV04_CMD_CLS *)
  ANDN %M92               (* VLV04_CMD_OPN *)
  IN
  OUT_BLK
  LD Q
  ST %M103                (* VLV04_TON_CLS_DN *)
  END_BLK
  // as ST:
  //   VLV04_TON_CLS(IN := VLV04_CMD_CLS AND NOT VLV04_CMD_OPN);
  //   VLV04_TON_CLS_DN := VLV04_TON_CLS.Q;

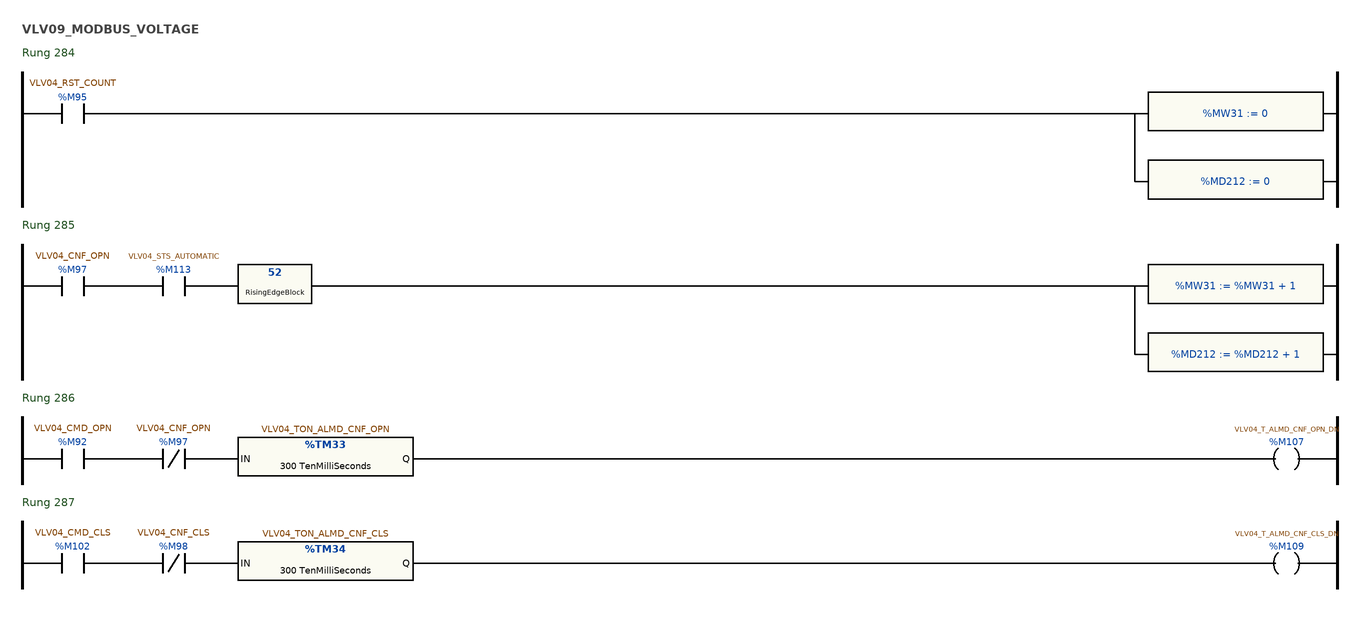

// Rung 284
  LD %M95                 (* VLV04_RST_COUNT *)
  [ %MW31 := 0 ]          (* VLV04_CNT_OPN_ACC *)
  [ %MD212 := 0 ]         (* VLV04_CNT_OPN_ACC2 *)
  // as ST:
  //   IF VLV04_RST_COUNT THEN VLV04_CNT_OPN_ACC := 0; END_IF;
  //   IF VLV04_RST_COUNT THEN VLV04_CNT_OPN_ACC2 := 0; END_IF;

// Rung 285
  LD %M97                 (* VLV04_CNF_OPN *)
  AND %M113               (* VLV04_STS_AUTOMATIC *)
  RISING52
  [ %MW31 := %MW31 + 1 ]  (* VLV04_CNT_OPN_ACC, VLV04_CNT_OPN_ACC *)
  [ %MD212 := %MD212 + 1 ](* VLV04_CNT_OPN_ACC2, VLV04_CNT_OPN_ACC2 *)
  // as ST:
  //   IF RISING(VLV04_CNF_OPN AND VLV04_STS_AUTOMATIC) THEN VLV04_CNT_OPN_ACC := VLV04_CNT_OPN_ACC + 1; END_IF;
  //   IF RISING(VLV04_CNF_OPN AND VLV04_STS_AUTOMATIC) THEN VLV04_CNT_OPN_ACC2 := VLV04_CNT_OPN_ACC2 + 1; END_IF;

// Rung 286
  BLK %TM33               (* VLV04_TON_ALMD_CNF_OPN *)
  LD %M92                 (* VLV04_CMD_OPN *)
  ANDN %M97               (* VLV04_CNF_OPN *)
  IN
  OUT_BLK
  LD Q
  ST %M107                (* VLV04_T_ALMD_CNF_OPN_DN *)
  END_BLK
  // as ST:
  //   VLV04_TON_ALMD_CNF_OPN(IN := VLV04_CMD_OPN AND NOT VLV04_CNF_OPN);
  //   VLV04_T_ALMD_CNF_OPN_DN := VLV04_TON_ALMD_CNF_OPN.Q;

// Rung 287
  BLK %TM34               (* VLV04_TON_ALMD_CNF_CLS *)
  LD %M102                (* VLV04_CMD_CLS *)
  ANDN %M98               (* VLV04_CNF_CLS *)
  IN
  OUT_BLK
  LD Q
  ST %M109                (* VLV04_T_ALMD_CNF_CLS_DN *)
  END_BLK
  // as ST:
  //   VLV04_TON_ALMD_CNF_CLS(IN := VLV04_CMD_CLS AND NOT VLV04_CNF_CLS);
  //   VLV04_T_ALMD_CNF_CLS_DN := VLV04_TON_ALMD_CNF_CLS.Q;

POU HORA
  (* SectionNumber=12 *)

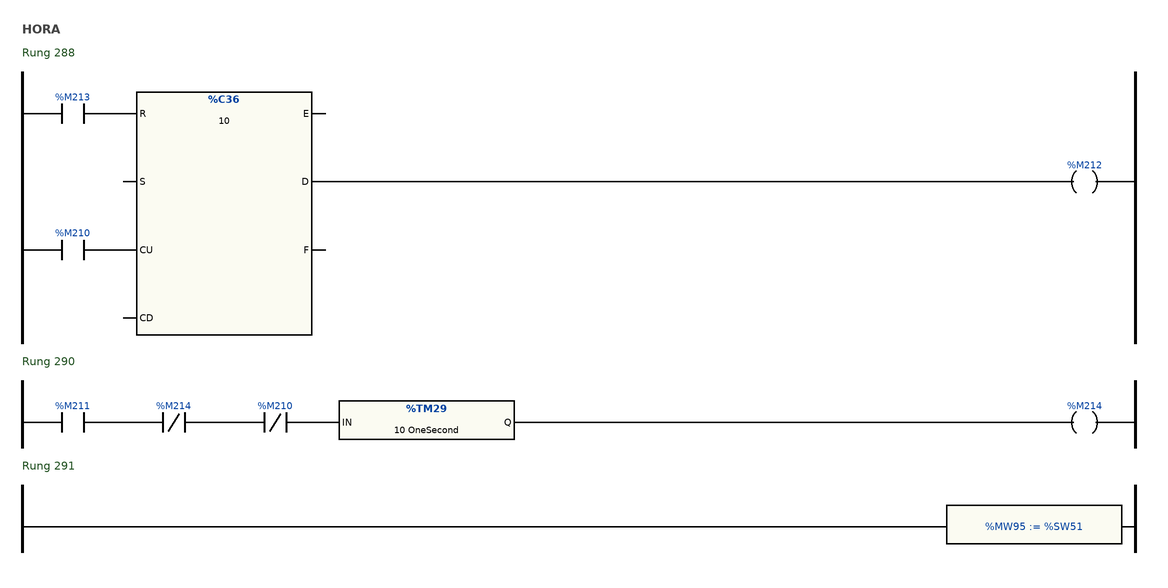

// Rung 288
  BLK %C36
  LD %M213
  R
  LD %M210
  CU
  OUT_BLK
  LD D
  ST %M212
  END_BLK
  // as ST:
  //   %C36(R := %M213, CU := %M210);
  //   %M212 := %C36.D;

// Rung 289
  BLK %C37
  LD 1
  AND( %M210
  OR %M213
  )
  R
  LD %M214
  CU
  OUT_BLK
  LD D
  ST %M210
  END_BLK
  // as ST:
  //   %C37(R := %M210 OR %M213, CU := %M214);
  //   %M210 := %C37.D;
  (* the ladder stored for this rung does not match its IL; not drawn *)

// Rung 290
  BLK %TM29
  LD %M211
  ANDN %M214
  ANDN %M210
  IN
  OUT_BLK
  LD Q
  ST %M214
  END_BLK
  // as ST:
  //   %TM29(IN := %M211 AND NOT %M214 AND NOT %M210);
  //   %M214 := %TM29.Q;

// Rung 291
  LD 1
  [ %MW95 := %SW51 ]      (* SW_RTCHHMM *)
  // as ST:
  //   %MW95 := SW_RTCHHMM;

Subroutine Get RTC
  (* SectionNumber=13, Number=0 *)

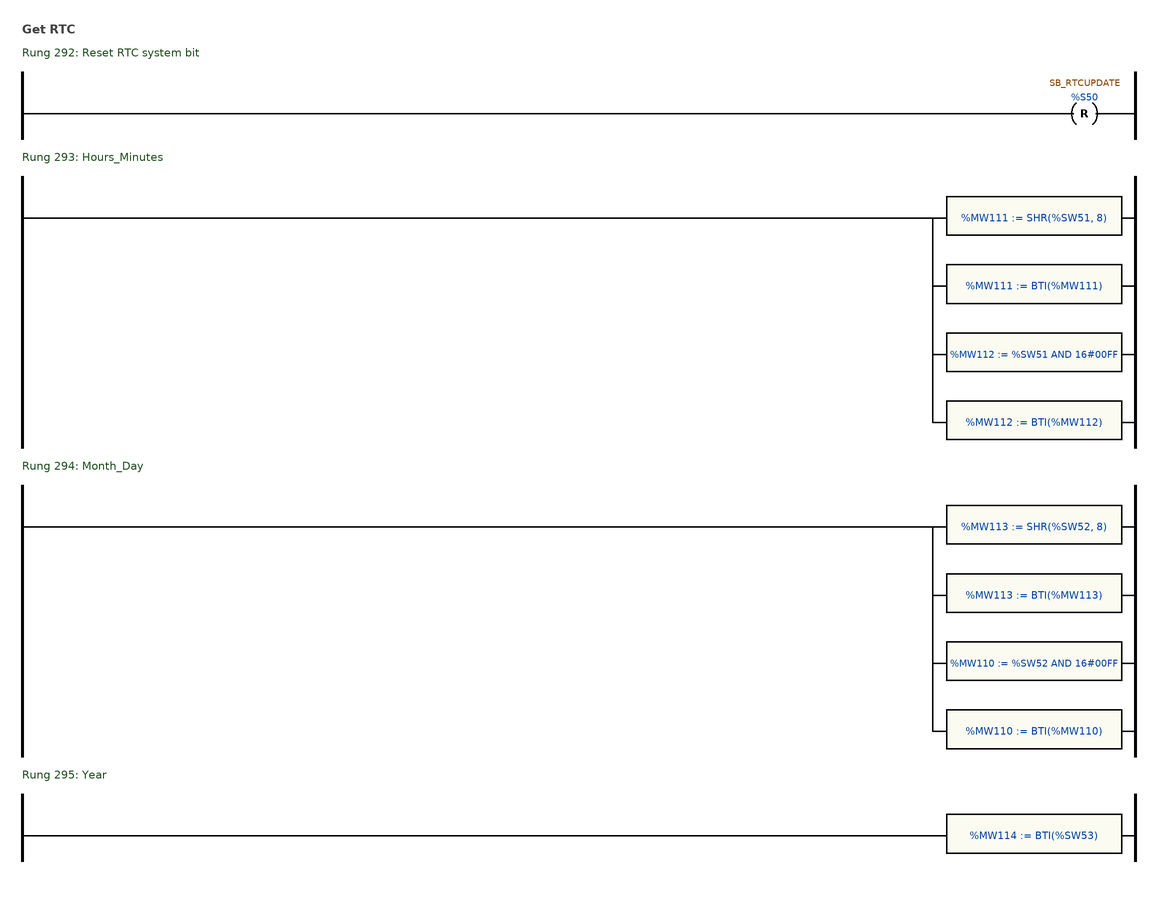

// Rung 292: Reset RTC system bit
  LD 1
  R %S50                  (* SB_RTCUPDATE *)
  // as ST:
  //   SB_RTCUPDATE := FALSE;

// Rung 293: Hours_Minutes
  LD 1
  [ %MW111 := SHR ( %SW51 , 8 ) ](* HOUR, SW_RTCHHMM *)
  [ %MW111 := BTI ( %MW111 ) ](* HOUR, HOUR *)
  [ %MW112 := %SW51 AND 16#00FF ](* MINUTES, SW_RTCHHMM *)
  [ %MW112 := BTI ( %MW112 ) ](* MINUTES, MINUTES *)
  // as ST:
  //   HOUR := SHR ( SW_RTCHHMM , 8 );
  //   HOUR := BTI ( HOUR );
  //   MINUTES := SW_RTCHHMM AND 16#00FF;
  //   MINUTES := BTI ( MINUTES );

// Rung 294: Month_Day
  LD 1
  [ %MW113 := SHR ( %SW52 , 8 ) ](* MONTH, SW_RTCMMDD *)
  [ %MW113 := BTI ( %MW113 ) ](* MONTH, MONTH *)
  [ %MW110 := %SW52 AND 16#00FF ](* DAY, SW_RTCMMDD *)
  [ %MW110 := BTI ( %MW110 ) ](* DAY, DAY *)
  // as ST:
  //   MONTH := SHR ( SW_RTCMMDD , 8 );
  //   MONTH := BTI ( MONTH );
  //   DAY := SW_RTCMMDD AND 16#00FF;
  //   DAY := BTI ( DAY );

// Rung 295: Year
  LD 1
  [ %MW114 := BTI ( %SW53 ) ](* YEAR, SW_RTCCCYY *)
  // as ST:
  //   YEAR := BTI ( SW_RTCCCYY );

Subroutine Free POU_0
  (* SectionNumber=14, Number=1 *)

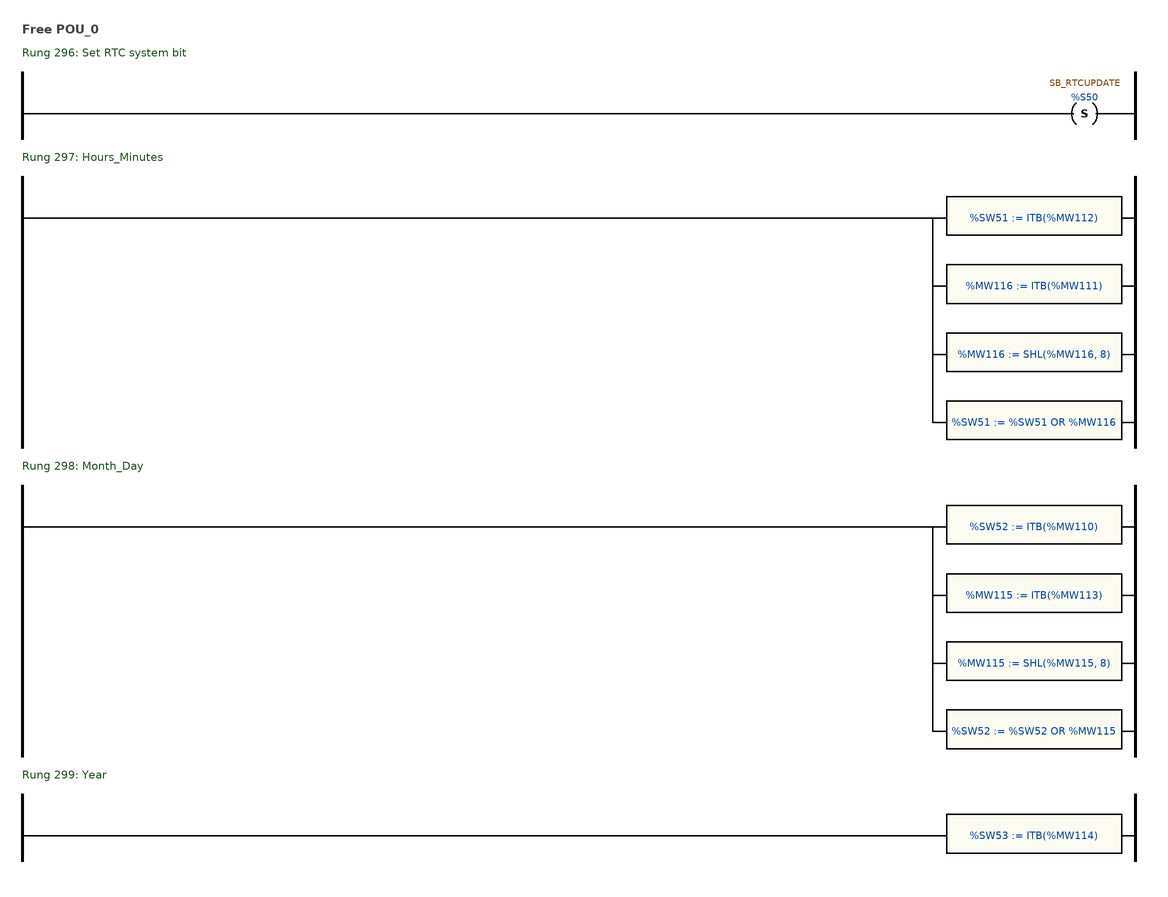

// Rung 296: Set RTC system bit
  LD 1
  S %S50                  (* SB_RTCUPDATE *)
  // as ST:
  //   SB_RTCUPDATE := TRUE;

// Rung 297: Hours_Minutes
  LD 1
  [ %SW51 := ITB ( %MW112 ) ](* SW_RTCHHMM, MINUTES *)
  [ %MW116 := ITB ( %MW111 ) ](* SCRAP_MINUTES, HOUR *)
  [ %MW116 := SHL ( %MW116 , 8 ) ](* SCRAP_MINUTES, SCRAP_MINUTES *)
  [ %SW51 := %SW51 OR %MW116 ](* SW_RTCHHMM, SW_RTCHHMM, SCRAP_MINUTES *)
  // as ST:
  //   SW_RTCHHMM := ITB ( MINUTES );
  //   SCRAP_MINUTES := ITB ( HOUR );
  //   SCRAP_MINUTES := SHL ( SCRAP_MINUTES , 8 );
  //   SW_RTCHHMM := SW_RTCHHMM OR SCRAP_MINUTES;

// Rung 298: Month_Day
  LD 1
  [ %SW52 := ITB ( %MW110 ) ](* SW_RTCMMDD, DAY *)
  [ %MW115 := ITB ( %MW113 ) ](* SCRAP_MONTH, MONTH *)
  [ %MW115 := SHL ( %MW115 , 8 ) ](* SCRAP_MONTH, SCRAP_MONTH *)
  [ %SW52 := %SW52 OR %MW115 ](* SW_RTCMMDD, SW_RTCMMDD, SCRAP_MONTH *)
  // as ST:
  //   SW_RTCMMDD := ITB ( DAY );
  //   SCRAP_MONTH := ITB ( MONTH );
  //   SCRAP_MONTH := SHL ( SCRAP_MONTH , 8 );
  //   SW_RTCMMDD := SW_RTCMMDD OR SCRAP_MONTH;

// Rung 299: Year
  LD 1
  [ %SW53 := ITB ( %MW114 ) ](* SW_RTCCCYY, YEAR *)
  // as ST:
  //   SW_RTCCCYY := ITB ( YEAR );
